    CONST robtarget Target_11220:=[[89.794609886,117.20347241,29.885035034],[0.692516726,0.060687774,-0.040025667,0.717729422],[0,0,0,0],[9E+09,9E+09,9E+09,9E+09,9E+09,9E+09]];
    CONST robtarget Target_11230:=[[90.590419724,116.924123639,29.863083326],[0.692516726,0.060687774,-0.040025666,0.717729422],[0,0,0,0],[9E+09,9E+09,9E+09,9E+09,9E+09,9E+09]];
    CONST robtarget Target_11240:=[[91.356578481,116.571453419,29.841743496],[0.692516726,0.060687774,-0.040025667,0.717729422],[0,0,0,0],[9E+09,9E+09,9E+09,9E+09,9E+09,9E+09]];
    CONST robtarget Target_11250:=[[92.086353126,116.148561032,29.821203079],[0.692516726,0.060687774,-0.040025667,0.717729422],[0,0,0,0],[9E+09,9E+09,9E+09,9E+09,9E+09,9E+09]];
    CONST robtarget Target_11260:=[[92.773330372,115.659162869,29.801642586],[0.692516726,0.060687774,-0.040025666,0.717729422],[0,0,0,0],[9E+09,9E+09,9E+09,9E+09,9E+09,9E+09]];
    CONST robtarget Target_11270:=[[93.411473041,115.107559779,29.783233914],[0.692516726,0.060687774,-0.040025667,0.717729422],[0,0,0,0],[9E+09,9E+09,9E+09,9E+09,9E+09,9E+09]];
    CONST robtarget Target_11280:=[[93.995173109,114.498599271,29.76613884],[0.692516726,0.060687774,-0.040025666,0.717729422],[0,0,0,0],[9E+09,9E+09,9E+09,9E+09,9E+09,9E+09]];
    CONST robtarget Target_11290:=[[94.519301002,113.837632911,29.750507595],[0.692516726,0.060687774,-0.040025667,0.717729422],[0,0,0,0],[9E+09,9E+09,9E+09,9E+09,9E+09,9E+09]];
    CONST robtarget Target_11300:=[[94.979250663,113.130469294,29.736477548],[0.692516726,0.060687774,-0.040025666,0.717729422],[0,0,0,0],[9E+09,9E+09,9E+09,9E+09,9E+09,9E+09]];
    CONST robtarget Target_11310:=[[95.370980037,112.383323003,29.724171995],[0.692516726,0.060687774,-0.040025666,0.717729422],[0,0,0,0],[9E+09,9E+09,9E+09,9E+09,9E+09,9E+09]];
    CONST robtarget Target_11320:=[[95.691046596,111.602759982,29.713699078],[0.692516726,0.060687774,-0.040025666,0.717729422],[0,0,0,0],[9E+09,9E+09,9E+09,9E+09,9E+09,9E+09]];
    CONST robtarget Target_11330:=[[95.93663758,110.79563985,29.705150834],[0.692516726,0.060687774,-0.040025666,0.717729422],[0,0,0,0],[9E+09,9E+09,9E+09,9E+09,9E+09,9E+09]];
    CONST robtarget Target_11340:=[[96.105594728,109.969055606,29.698602383],[0.692516726,0.060687774,-0.040025667,0.717729422],[0,0,0,0],[9E+09,9E+09,9E+09,9E+09,9E+09,9E+09]];
    CONST robtarget Target_11350:=[[96.196433238,109.130271302,29.694111275],[0.692516726,0.060687774,-0.040025667,0.717729422],[0,0,0,0],[9E+09,9E+09,9E+09,9E+09,9E+09,9E+09]];
    CONST robtarget Target_11360:=[[96.208354819,108.286658206,29.691716978],[0.692516726,0.060687774,-0.040025667,0.717729422],[0,0,0,0],[9E+09,9E+09,9E+09,9E+09,9E+09,9E+09]];
    CONST robtarget Target_11370:=[[96.141254703,107.445630019,29.691440532],[0.692516726,0.060687774,-0.040025667,0.717729422],[0,0,0,0],[9E+09,9E+09,9E+09,9E+09,9E+09,9E+09]];
    CONST robtarget Target_11380:=[[95.995722568,106.614577729,29.693284368],[0.692516726,0.060687774,-0.040025667,0.717729422],[0,0,0,0],[9E+09,9E+09,9E+09,9E+09,9E+09,9E+09]];
    CONST robtarget Target_11390:=[[95.773037356,105.80080465,29.697232281],[0.692516726,0.060687774,-0.040025667,0.717729422],[0,0,0,0],[9E+09,9E+09,9E+09,9E+09,9E+09,9E+09]];
    CONST robtarget Target_11400:=[[95.475156032,105.011462252,29.703249576],[0.692516726,0.060687774,-0.040025667,0.717729422],[0,0,0,0],[9E+09,9E+09,9E+09,9E+09,9E+09,9E+09]];
    CONST robtarget Target_11410:=[[95.104696388,104.253487303,29.711283375],[0.692516726,0.060687774,-0.040025666,0.717729422],[0,0,0,0],[9E+09,9E+09,9E+09,9E+09,9E+09,9E+09]];
    CONST robtarget Target_11420:=[[94.664914038,103.533540915,29.721263075],[0.692516726,0.060687774,-0.040025667,0.717729422],[0,0,0,0],[9E+09,9E+09,9E+09,9E+09,9E+09,9E+09]];
    CONST robtarget Target_11430:=[[94.159673804,102.857950002,29.733100975],[0.692516726,0.060687774,-0.040025667,0.717729422],[0,0,0,0],[9E+09,9E+09,9E+09,9E+09,9E+09,9E+09]];
    CONST robtarget Target_11440:=[[93.593415754,102.232651681,29.746693042],[0.692516726,0.060687774,-0.040025667,0.717729422],[0,0,0,0],[9E+09,9E+09,9E+09,9E+09,9E+09,9E+09]];
    CONST robtarget Target_11450:=[[92.971116187,101.663141097,29.761919829],[0.692516726,0.060687774,-0.040025666,0.717729422],[0,0,0,0],[9E+09,9E+09,9E+09,9E+09,9E+09,9E+09]];
    CONST robtarget Target_11460:=[[92.298243892,101.154423128,29.778647523],[0.692516726,0.060687774,-0.040025667,0.717729422],[0,0,0,0],[9E+09,9E+09,9E+09,9E+09,9E+09,9E+09]];
    CONST robtarget Target_11470:=[[91.580712095,100.710968408,29.79672912],[0.692516726,0.060687774,-0.040025667,0.717729422],[0,0,0,0],[9E+09,9E+09,9E+09,9E+09,9E+09,9E+09]];
    CONST robtarget Target_11480:=[[90.824826492,100.336674031,29.816005718],[0.692516726,0.060687774,-0.040025667,0.717729422],[0,0,0,0],[9E+09,9E+09,9E+09,9E+09,9E+09,9E+09]];
    CONST robtarget Target_11490:=[[90.037229833,100.034829312,29.836307913],[0.692516726,0.060687774,-0.040025667,0.717729422],[0,0,0,0],[9E+09,9E+09,9E+09,9E+09,9E+09,9E+09]];
    CONST robtarget Target_11500:=[[89.224843544,99.808086869,29.85745729],[0.692516726,0.060687774,-0.040025666,0.717729422],[0,0,0,0],[9E+09,9E+09,9E+09,9E+09,9E+09,9E+09]];
    CONST robtarget Target_11510:=[[88.394806907,99.658439327,29.879267987],[0.692516726,0.060687774,-0.040025666,0.717729422],[0,0,0,0],[9E+09,9E+09,9E+09,9E+09,9E+09,9E+09]];
    CONST robtarget Target_11520:=[[87.554414313,99.587201792,29.901548331],[0.692516726,0.060687774,-0.040025667,0.717729422],[0,0,0,0],[9E+09,9E+09,9E+09,9E+09,9E+09,9E+09]];
    CONST robtarget Target_11530:=[[86.753090736,99.66099158,-0.087656987],[0.692516726,0.060687774,-0.040025667,0.717729422],[0,0,0,0],[9E+09,9E+09,9E+09,9E+09,9E+09,9E+09]];
    CONST robtarget Target_11540:=[[119.551173325,78.726504599,-1.015545136],[0.692516726,0.060687774,-0.040025666,0.717729422],[0,0,0,0],[9E+09,9E+09,9E+09,9E+09,9E+09,9E+09]];
    CONST robtarget Target_11550:=[[120.352496902,78.652714811,28.973660182],[0.692516726,0.060687774,-0.040025666,0.717729422],[0,0,0,0],[9E+09,9E+09,9E+09,9E+09,9E+09,9E+09]];
    CONST robtarget Target_11560:=[[120.164706446,83.64915705,28.990971989],[0.692516726,0.060687774,-0.040025666,0.717729422],[0,0,0,0],[9E+09,9E+09,9E+09,9E+09,9E+09,9E+09]];
    CONST robtarget Target_11570:=[[110.175332474,83.272786458,29.256965985],[0.692516726,0.060687774,-0.040025666,0.717729422],[0,0,0,0],[9E+09,9E+09,9E+09,9E+09,9E+09,9E+09]];
    CONST robtarget Target_11580:=[[110.363122929,78.276344219,29.239654179],[0.692516726,0.060687774,-0.040025666,0.717729422],[0,0,0,0],[9E+09,9E+09,9E+09,9E+09,9E+09,9E+09]];
    CONST robtarget Target_11590:=[[120.352496902,78.652714811,28.973660182],[0.692516726,0.060687774,-0.040025666,0.717729422],[0,0,0,0],[9E+09,9E+09,9E+09,9E+09,9E+09,9E+09]];
    CONST robtarget Target_11600:=[[119.551173325,78.726504599,-1.015545136],[0.692516726,0.060687774,-0.040025666,0.717729422],[0,0,0,0],[9E+09,9E+09,9E+09,9E+09,9E+09,9E+09]];
    CONST robtarget Target_11610:=[[94.577738392,77.785578119,-0.350560144],[0.692516726,0.060687774,-0.040025666,0.717729422],[0,0,0,0],[9E+09,9E+09,9E+09,9E+09,9E+09,9E+09]];
    CONST robtarget Target_11620:=[[95.379061969,77.711788331,29.638645173],[0.692516726,0.060687774,-0.040025666,0.717729422],[0,0,0,0],[9E+09,9E+09,9E+09,9E+09,9E+09,9E+09]];
    CONST robtarget Target_11630:=[[105.368435942,78.088158923,29.372651177],[0.692516726,0.060687774,-0.040025666,0.717729422],[0,0,0,0],[9E+09,9E+09,9E+09,9E+09,9E+09,9E+09]];
    CONST robtarget Target_11640:=[[105.180645487,83.084601162,29.389962984],[0.692516726,0.060687774,-0.040025666,0.717729422],[0,0,0,0],[9E+09,9E+09,9E+09,9E+09,9E+09,9E+09]];
    CONST robtarget Target_11650:=[[95.191271514,82.70823057,29.65595698],[0.692516726,0.060687774,-0.040025666,0.717729422],[0,0,0,0],[9E+09,9E+09,9E+09,9E+09,9E+09,9E+09]];
    CONST robtarget Target_11660:=[[95.379061969,77.711788331,29.638645173],[0.692516726,0.060687774,-0.040025666,0.717729422],[0,0,0,0],[9E+09,9E+09,9E+09,9E+09,9E+09,9E+09]];
    CONST robtarget Target_11670:=[[94.577738392,77.785578119,-0.350560144],[0.692516726,0.060687774,-0.040025666,0.717729422],[0,0,0,0],[9E+09,9E+09,9E+09,9E+09,9E+09,9E+09]];
    CONST robtarget Target_11680:=[[89.583051406,77.597392823,-0.217563146],[0.692516726,0.060687774,-0.040025666,0.717729422],[0,0,0,0],[9E+09,9E+09,9E+09,9E+09,9E+09,9E+09]];
    CONST robtarget Target_11690:=[[90.384374983,77.523603036,29.771642172],[0.692516726,0.060687774,-0.040025666,0.717729422],[0,0,0,0],[9E+09,9E+09,9E+09,9E+09,9E+09,9E+09]];
    CONST robtarget Target_11700:=[[90.196584528,82.520045274,29.788953979],[0.692516726,0.060687774,-0.040025666,0.717729422],[0,0,0,0],[9E+09,9E+09,9E+09,9E+09,9E+09,9E+09]];
    CONST robtarget Target_11710:=[[80.207210555,82.143674683,30.054947975],[0.692516726,0.060687774,-0.040025666,0.717729422],[0,0,0,0],[9E+09,9E+09,9E+09,9E+09,9E+09,9E+09]];
    CONST robtarget Target_11720:=[[80.39500101,77.147232444,30.037636168],[0.692516726,0.060687774,-0.040025666,0.717729422],[0,0,0,0],[9E+09,9E+09,9E+09,9E+09,9E+09,9E+09]];
    CONST robtarget Target_11730:=[[90.384374983,77.523603036,29.771642172],[0.692516726,0.060687774,-0.040025666,0.717729422],[0,0,0,0],[9E+09,9E+09,9E+09,9E+09,9E+09,9E+09]];
    CONST robtarget Target_11740:=[[89.583051406,77.597392823,-0.217563146],[0.692516726,0.060687774,-0.040025666,0.717729422],[0,0,0,0],[9E+09,9E+09,9E+09,9E+09,9E+09,9E+09]];






    CONST jointtarget Home_ABS:= [[0,0,0,0,30,0],[9E+09,9E+09,9E+09,9E+09,9E+09,9E+09]];
    CONST jointtarget Mantenimiento_Point:= [[90,0,0,0,30,0],[9E+09,9E+09,9E+09,9E+09,9E+09,9E+09]];
    !***********************************************************
    !
    ! M?dulo:  Module1
    !
    ! Descripción:
    !   <Introduzca la descripción aquí>
    !
    ! Autor: pache
    !
    ! Versión: 1.0
    !
    !***********************************************************


    !***********************************************************
    !
    ! Procedimiento Main
    !
    !   Este es el punto de entrada de su programa
    !
PROC main()

        ! Limpiamos la pantalla del control virtual
        TPErase;
        TPWrite "SISTEMA INICIADO";

        MoveAbsJ Home_ABS, v300, z1, tool0;

        TPWrite "INICIO PROGRAMA";
        TPWrite "APAGADO BANDA TRANASPORTADORA";
        Reset DO_02;
        Reset DO_01;
        RESET BWD_Conveyor;
        RESET FWD_Conveyor;




        ! 1. Apagamos la banda por seguridad al arrancar

        WHILE TRUE DO

            IF DI_03 = 1 THEN
                Set BWD_Conveyor;
                WaitTime 4.275;
                Reset FWD_Conveyor;
                Reset BWD_Conveyor;
            ENDIF


            TPWrite "ESPERANDO QUE PRESIONE DI_01...";
            ! 2. Esperamos el botón de inicio
            IF DI_01 = 1 AND DI_02 = 0 THEN




                    TPWrite "MOVIENDO CAJA...";

                    ! 3. Encendemos la banda
                    set FWD_Conveyor;
                    set DO_01;

                    ! 4. Tiempo de viaje (ajustado a tu prueba)
                    WaitTime 4.275;

                    ! 5. Detenemos la caja
                    Reset FWD_Conveyor;
                    TPWrite "CAJA EN POSICION - INICIANDO GRABADO";

                    ! --------------------------------------------------------
                    ! 6. LLAMADA A LAS TRAYECTORIAS
                    Path_aprox;
                    WaitTime 1;
                    Path_duvan;
                    Path_mora;
                    Path_gusta;
                    Path_robot;
                    Path_220;
                    WaitTime 2;
                    Path_home;
                    WaitTime 5;
                    reset DO_01;

                ELSEIF DI_01 = 0 AND DI_02=1 THEN
                Set DO_02;
                TPWrite "RUTINA CAMBIO DE HERRAMIENTA";
                MoveAbsJ Mantenimiento_Point,v100,z1,tool0;
                TPWrite "PELIGRO";
                TPWrite "OPERARIO CERCA A HERRAMIENTA";
                TPWrite "PRESIONE LOS DOS BOTONES PARA CONTINUAR EL PROGRAMA";
                WaitDI DI_01,1;
                WaitDI DI_02,1;
                Reset DO_02;
                TPWrite "REANUDANDO PROGRAMA";
                WaitTime 3;
                MoveAbsJ Home_ABS,v100,z1,tool0;
                ELSEIF DI_01 = 0 AND DI_02=0 THEN
                TPWrite "ESPERANDO INSTRUCCIÓNES";
                ELSEIF DI_01 = 1 AND DI_02=1 THEN
                TPWrite "ERROR";
                TPWrite "NO DEBE PRESIONAR AMBAS ENTRADAS AL TIEMPO";
            ENDIF

            TPWrite "CICLO TERMINADO. MUEVA LA CAJA AL INICIO.";
        ENDWHILE
        WaitTime 1.0;
    ENDPROC




    PROC Path_aprox()
        MoveL Target_home,v100,z1,MarcadorVirtual\WObj:=wobj0;
        MoveL Target_aprox1,v100,z1,MarcadorVirtual\WObj:=wobj0;
        MoveL Target_aprox2,v100,z1,MarcadorVirtual\WObj:=wobj0;

    ENDPROC
    PROC Path_10()
        MoveL Target_aprox2,v60,z1,MarcadorVirtual\WObj:=wobj0;
        MoveL Target_10,v60,z1,MarcadorVirtual\WObj:=wobj_JMora;
    ENDPROC
    PROC Path_20()
        MoveL Target_540,v60,z1,MarcadorVirtual\WObj:=wobj_JMora;
        MoveL Target_550,v60,z1,MarcadorVirtual\WObj:=wobj_JMora;
    ENDPROC
    PROC Path_home()
        MoveL Target_home,v100,z1,MarcadorVirtual\WObj:=wobj0;
    ENDPROC
    PROC Path_30()
        MoveL Target_1070,v60,z1,MarcadorVirtual\WObj:=wobj_JMora;
        MoveL Target_1080,v60,z1,MarcadorVirtual\WObj:=wobj_JMora;
    ENDPROC
    PROC Path_40()
        MoveL Target_1560,v60,z1,MarcadorVirtual\WObj:=wobj_JMora;
        MoveL Target_1570,v60,z1,MarcadorVirtual\WObj:=wobj_JMora;
    ENDPROC
    PROC Path_50()
        MoveL Target_2360,v60,z1,MarcadorVirtual\WObj:=wobj_JMora;
        MoveL Target_2370,v60,z1,MarcadorVirtual\WObj:=wobj_JMora;
    ENDPROC
    PROC Path_60()
        MoveL Target_1070,v60,z1,MarcadorVirtual\WObj:=wobj_JMora;
        MoveL Target_1080,v60,z1,MarcadorVirtual\WObj:=wobj_JMora;
    ENDPROC
    PROC Path_D()
        MoveL Target_10,v60,z1,MarcadorVirtual\WObj:=wobj_JMora;
        MoveL Target_20,v60,z1,MarcadorVirtual\WObj:=wobj_JMora;
        MoveL Target_30,v60,z1,MarcadorVirtual\WObj:=wobj_JMora;
        MoveL Target_40,v60,z1,MarcadorVirtual\WObj:=wobj_JMora;
        MoveL Target_50,v60,z1,MarcadorVirtual\WObj:=wobj_JMora;
        MoveL Target_60,v60,z1,MarcadorVirtual\WObj:=wobj_JMora;
        MoveL Target_70,v60,z1,MarcadorVirtual\WObj:=wobj_JMora;
        MoveL Target_80,v60,z1,MarcadorVirtual\WObj:=wobj_JMora;
        MoveL Target_90,v60,z1,MarcadorVirtual\WObj:=wobj_JMora;
        MoveL Target_100,v60,z1,MarcadorVirtual\WObj:=wobj_JMora;
        MoveL Target_110,v60,z1,MarcadorVirtual\WObj:=wobj_JMora;
        MoveL Target_120,v60,z1,MarcadorVirtual\WObj:=wobj_JMora;
        MoveL Target_130,v60,z1,MarcadorVirtual\WObj:=wobj_JMora;
        MoveL Target_140,v60,z1,MarcadorVirtual\WObj:=wobj_JMora;
        MoveL Target_150,v60,z1,MarcadorVirtual\WObj:=wobj_JMora;
        MoveL Target_160,v60,z1,MarcadorVirtual\WObj:=wobj_JMora;
        MoveL Target_170,v60,z1,MarcadorVirtual\WObj:=wobj_JMora;
        MoveL Target_180,v60,z1,MarcadorVirtual\WObj:=wobj_JMora;
        MoveL Target_190,v60,z1,MarcadorVirtual\WObj:=wobj_JMora;
        MoveL Target_200,v60,z1,MarcadorVirtual\WObj:=wobj_JMora;
        MoveL Target_210,v60,z1,MarcadorVirtual\WObj:=wobj_JMora;
        MoveL Target_220,v60,z1,MarcadorVirtual\WObj:=wobj_JMora;
        MoveL Target_230,v60,z1,MarcadorVirtual\WObj:=wobj_JMora;
        MoveL Target_240,v60,z1,MarcadorVirtual\WObj:=wobj_JMora;
        MoveL Target_250,v60,z1,MarcadorVirtual\WObj:=wobj_JMora;
        MoveL Target_260,v60,z1,MarcadorVirtual\WObj:=wobj_JMora;
        MoveL Target_270,v60,z1,MarcadorVirtual\WObj:=wobj_JMora;
        MoveL Target_280,v60,z1,MarcadorVirtual\WObj:=wobj_JMora;
        MoveL Target_290,v60,z1,MarcadorVirtual\WObj:=wobj_JMora;
        MoveL Target_300,v60,z1,MarcadorVirtual\WObj:=wobj_JMora;
        MoveL Target_310,v60,z1,MarcadorVirtual\WObj:=wobj_JMora;
        MoveL Target_320,v60,z1,MarcadorVirtual\WObj:=wobj_JMora;
        MoveL Target_330,v60,z1,MarcadorVirtual\WObj:=wobj_JMora;
        MoveL Target_340,v60,z1,MarcadorVirtual\WObj:=wobj_JMora;
        MoveL Target_350,v60,z1,MarcadorVirtual\WObj:=wobj_JMora;
        MoveL Target_360,v60,z1,MarcadorVirtual\WObj:=wobj_JMora;
        MoveL Target_370,v60,z1,MarcadorVirtual\WObj:=wobj_JMora;
        MoveL Target_380,v60,z1,MarcadorVirtual\WObj:=wobj_JMora;
        MoveL Target_390,v60,z1,MarcadorVirtual\WObj:=wobj_JMora;
        MoveL Target_400,v60,z1,MarcadorVirtual\WObj:=wobj_JMora;
        MoveL Target_410,v60,z1,MarcadorVirtual\WObj:=wobj_JMora;
        MoveL Target_420,v60,z1,MarcadorVirtual\WObj:=wobj_JMora;
        MoveL Target_430,v60,z1,MarcadorVirtual\WObj:=wobj_JMora;
        MoveL Target_440,v60,z1,MarcadorVirtual\WObj:=wobj_JMora;
        MoveL Target_450,v60,z1,MarcadorVirtual\WObj:=wobj_JMora;
        MoveL Target_460,v60,z1,MarcadorVirtual\WObj:=wobj_JMora;
        MoveL Target_470,v60,z1,MarcadorVirtual\WObj:=wobj_JMora;
        MoveL Target_480,v60,z1,MarcadorVirtual\WObj:=wobj_JMora;
        MoveL Target_490,v60,z1,MarcadorVirtual\WObj:=wobj_JMora;
        MoveL Target_500,v60,z1,MarcadorVirtual\WObj:=wobj_JMora;
        MoveL Target_510,v60,z1,MarcadorVirtual\WObj:=wobj_JMora;
        MoveL Target_520,v60,z1,MarcadorVirtual\WObj:=wobj_JMora;
        MoveL Target_530,v60,z1,MarcadorVirtual\WObj:=wobj_JMora;
        MoveL Target_540,v60,z1,MarcadorVirtual\WObj:=wobj_JMora;
    ENDPROC
    PROC Path_U1()
        MoveL Target_550,v60,z1,MarcadorVirtual\WObj:=wobj_JMora;
        MoveL Target_560,v60,z1,MarcadorVirtual\WObj:=wobj_JMora;
        MoveL Target_570,v60,z1,MarcadorVirtual\WObj:=wobj_JMora;
        MoveL Target_580,v60,z1,MarcadorVirtual\WObj:=wobj_JMora;
        MoveL Target_590,v60,z1,MarcadorVirtual\WObj:=wobj_JMora;
        MoveL Target_600,v60,z1,MarcadorVirtual\WObj:=wobj_JMora;
        MoveL Target_610,v60,z1,MarcadorVirtual\WObj:=wobj_JMora;
        MoveL Target_620,v60,z1,MarcadorVirtual\WObj:=wobj_JMora;
        MoveL Target_630,v60,z1,MarcadorVirtual\WObj:=wobj_JMora;
        MoveL Target_640,v60,z1,MarcadorVirtual\WObj:=wobj_JMora;
        MoveL Target_650,v60,z1,MarcadorVirtual\WObj:=wobj_JMora;
        MoveL Target_660,v60,z1,MarcadorVirtual\WObj:=wobj_JMora;
        MoveL Target_670,v60,z1,MarcadorVirtual\WObj:=wobj_JMora;
        MoveL Target_680,v60,z1,MarcadorVirtual\WObj:=wobj_JMora;
        MoveL Target_690,v60,z1,MarcadorVirtual\WObj:=wobj_JMora;
        MoveL Target_700,v60,z1,MarcadorVirtual\WObj:=wobj_JMora;
        MoveL Target_710,v60,z1,MarcadorVirtual\WObj:=wobj_JMora;
        MoveL Target_720,v60,z1,MarcadorVirtual\WObj:=wobj_JMora;
        MoveL Target_730,v60,z1,MarcadorVirtual\WObj:=wobj_JMora;
        MoveL Target_740,v60,z1,MarcadorVirtual\WObj:=wobj_JMora;
        MoveL Target_750,v60,z1,MarcadorVirtual\WObj:=wobj_JMora;
        MoveL Target_760,v60,z1,MarcadorVirtual\WObj:=wobj_JMora;
        MoveL Target_770,v60,z1,MarcadorVirtual\WObj:=wobj_JMora;
        MoveL Target_780,v60,z1,MarcadorVirtual\WObj:=wobj_JMora;
        MoveL Target_790,v60,z1,MarcadorVirtual\WObj:=wobj_JMora;
        MoveL Target_800,v60,z1,MarcadorVirtual\WObj:=wobj_JMora;
        MoveL Target_810,v60,z1,MarcadorVirtual\WObj:=wobj_JMora;
        MoveL Target_820,v60,z1,MarcadorVirtual\WObj:=wobj_JMora;
        MoveL Target_830,v60,z1,MarcadorVirtual\WObj:=wobj_JMora;
        MoveL Target_840,v60,z1,MarcadorVirtual\WObj:=wobj_JMora;
        MoveL Target_850,v60,z1,MarcadorVirtual\WObj:=wobj_JMora;
        MoveL Target_860,v60,z1,MarcadorVirtual\WObj:=wobj_JMora;
        MoveL Target_870,v60,z1,MarcadorVirtual\WObj:=wobj_JMora;
        MoveL Target_880,v60,z1,MarcadorVirtual\WObj:=wobj_JMora;
        MoveL Target_890,v60,z1,MarcadorVirtual\WObj:=wobj_JMora;
        MoveL Target_900,v60,z1,MarcadorVirtual\WObj:=wobj_JMora;
        MoveL Target_910,v60,z1,MarcadorVirtual\WObj:=wobj_JMora;
        MoveL Target_920,v60,z1,MarcadorVirtual\WObj:=wobj_JMora;
        MoveL Target_930,v60,z1,MarcadorVirtual\WObj:=wobj_JMora;
        MoveL Target_940,v60,z1,MarcadorVirtual\WObj:=wobj_JMora;
        MoveL Target_950,v60,z1,MarcadorVirtual\WObj:=wobj_JMora;
        MoveL Target_960,v60,z1,MarcadorVirtual\WObj:=wobj_JMora;
        MoveL Target_970,v60,z1,MarcadorVirtual\WObj:=wobj_JMora;
        MoveL Target_980,v60,z1,MarcadorVirtual\WObj:=wobj_JMora;
        MoveL Target_990,v60,z1,MarcadorVirtual\WObj:=wobj_JMora;
        MoveL Target_1000,v60,z1,MarcadorVirtual\WObj:=wobj_JMora;
        MoveL Target_1010,v60,z1,MarcadorVirtual\WObj:=wobj_JMora;
        MoveL Target_1020,v60,z1,MarcadorVirtual\WObj:=wobj_JMora;
        MoveL Target_1030,v60,z1,MarcadorVirtual\WObj:=wobj_JMora;
        MoveL Target_1040,v60,z1,MarcadorVirtual\WObj:=wobj_JMora;
        MoveL Target_1050,v60,z1,MarcadorVirtual\WObj:=wobj_JMora;
        MoveL Target_1060,v60,z1,MarcadorVirtual\WObj:=wobj_JMora;
        MoveL Target_1070,v60,z1,MarcadorVirtual\WObj:=wobj_JMora;
    ENDPROC
    PROC Path_V()
        MoveL Target_1080,v60,z1,MarcadorVirtual\WObj:=wobj_JMora;
        MoveL Target_1090,v60,z1,MarcadorVirtual\WObj:=wobj_JMora;
        MoveL Target_1100,v60,z1,MarcadorVirtual\WObj:=wobj_JMora;
        MoveL Target_1110,v60,z1,MarcadorVirtual\WObj:=wobj_JMora;
        MoveL Target_1120,v60,z1,MarcadorVirtual\WObj:=wobj_JMora;
        MoveL Target_1130,v60,z1,MarcadorVirtual\WObj:=wobj_JMora;
        MoveL Target_1140,v60,z1,MarcadorVirtual\WObj:=wobj_JMora;
        MoveL Target_1150,v60,z1,MarcadorVirtual\WObj:=wobj_JMora;
        MoveL Target_1160,v60,z1,MarcadorVirtual\WObj:=wobj_JMora;
        MoveL Target_1170,v60,z1,MarcadorVirtual\WObj:=wobj_JMora;
        MoveL Target_1180,v60,z1,MarcadorVirtual\WObj:=wobj_JMora;
        MoveL Target_1190,v60,z1,MarcadorVirtual\WObj:=wobj_JMora;
        MoveL Target_1200,v60,z1,MarcadorVirtual\WObj:=wobj_JMora;
        MoveL Target_1210,v60,z1,MarcadorVirtual\WObj:=wobj_JMora;
        MoveL Target_1220,v60,z1,MarcadorVirtual\WObj:=wobj_JMora;
        MoveL Target_1230,v60,z1,MarcadorVirtual\WObj:=wobj_JMora;
        MoveL Target_1240,v60,z1,MarcadorVirtual\WObj:=wobj_JMora;
        MoveL Target_1250,v60,z1,MarcadorVirtual\WObj:=wobj_JMora;
        MoveL Target_1260,v60,z1,MarcadorVirtual\WObj:=wobj_JMora;
        MoveL Target_1270,v60,z1,MarcadorVirtual\WObj:=wobj_JMora;
        MoveL Target_1280,v60,z1,MarcadorVirtual\WObj:=wobj_JMora;
        MoveL Target_1290,v60,z1,MarcadorVirtual\WObj:=wobj_JMora;
        MoveL Target_1300,v60,z1,MarcadorVirtual\WObj:=wobj_JMora;
        MoveL Target_1310,v60,z1,MarcadorVirtual\WObj:=wobj_JMora;
        MoveL Target_1320,v60,z1,MarcadorVirtual\WObj:=wobj_JMora;
        MoveL Target_1330,v60,z1,MarcadorVirtual\WObj:=wobj_JMora;
        MoveL Target_1340,v60,z1,MarcadorVirtual\WObj:=wobj_JMora;
        MoveL Target_1350,v60,z1,MarcadorVirtual\WObj:=wobj_JMora;
        MoveL Target_1360,v60,z1,MarcadorVirtual\WObj:=wobj_JMora;
        MoveL Target_1370,v60,z1,MarcadorVirtual\WObj:=wobj_JMora;
        MoveL Target_1380,v60,z1,MarcadorVirtual\WObj:=wobj_JMora;
        MoveL Target_1390,v60,z1,MarcadorVirtual\WObj:=wobj_JMora;
        MoveL Target_1400,v60,z1,MarcadorVirtual\WObj:=wobj_JMora;
        MoveL Target_1410,v60,z1,MarcadorVirtual\WObj:=wobj_JMora;
        MoveL Target_1420,v60,z1,MarcadorVirtual\WObj:=wobj_JMora;
        MoveL Target_1430,v60,z1,MarcadorVirtual\WObj:=wobj_JMora;
        MoveL Target_1440,v60,z1,MarcadorVirtual\WObj:=wobj_JMora;
        MoveL Target_1450,v60,z1,MarcadorVirtual\WObj:=wobj_JMora;
        MoveL Target_1460,v60,z1,MarcadorVirtual\WObj:=wobj_JMora;
        MoveL Target_1470,v60,z1,MarcadorVirtual\WObj:=wobj_JMora;
        MoveL Target_1480,v60,z1,MarcadorVirtual\WObj:=wobj_JMora;
        MoveL Target_1490,v60,z1,MarcadorVirtual\WObj:=wobj_JMora;
        MoveL Target_1500,v60,z1,MarcadorVirtual\WObj:=wobj_JMora;
        MoveL Target_1510,v60,z1,MarcadorVirtual\WObj:=wobj_JMora;
        MoveL Target_1520,v60,z1,MarcadorVirtual\WObj:=wobj_JMora;
        MoveL Target_1530,v60,z1,MarcadorVirtual\WObj:=wobj_JMora;
        MoveL Target_1540,v60,z1,MarcadorVirtual\WObj:=wobj_JMora;
        MoveL Target_1550,v60,z1,MarcadorVirtual\WObj:=wobj_JMora;
        MoveL Target_1560,v60,z1,MarcadorVirtual\WObj:=wobj_JMora;
    ENDPROC
    PROC Path_A1()
        MoveL Target_1570,v60,z1,MarcadorVirtual\WObj:=wobj_JMora;
        MoveL Target_1580,v60,z1,MarcadorVirtual\WObj:=wobj_JMora;
        MoveL Target_1590,v60,z1,MarcadorVirtual\WObj:=wobj_JMora;
        MoveL Target_1600,v60,z1,MarcadorVirtual\WObj:=wobj_JMora;
        MoveL Target_1610,v60,z1,MarcadorVirtual\WObj:=wobj_JMora;
        MoveL Target_1620,v60,z1,MarcadorVirtual\WObj:=wobj_JMora;
        MoveL Target_1630,v60,z1,MarcadorVirtual\WObj:=wobj_JMora;
        MoveL Target_1640,v60,z1,MarcadorVirtual\WObj:=wobj_JMora;
        MoveL Target_1650,v60,z1,MarcadorVirtual\WObj:=wobj_JMora;
        MoveL Target_1660,v60,z1,MarcadorVirtual\WObj:=wobj_JMora;
        MoveL Target_1670,v60,z1,MarcadorVirtual\WObj:=wobj_JMora;
        MoveL Target_1680,v60,z1,MarcadorVirtual\WObj:=wobj_JMora;
        MoveL Target_1690,v60,z1,MarcadorVirtual\WObj:=wobj_JMora;
        MoveL Target_1700,v60,z1,MarcadorVirtual\WObj:=wobj_JMora;
        MoveL Target_1710,v60,z1,MarcadorVirtual\WObj:=wobj_JMora;
        MoveL Target_1720,v60,z1,MarcadorVirtual\WObj:=wobj_JMora;
        MoveL Target_1730,v60,z1,MarcadorVirtual\WObj:=wobj_JMora;
        MoveL Target_1740,v60,z1,MarcadorVirtual\WObj:=wobj_JMora;
        MoveL Target_1750,v60,z1,MarcadorVirtual\WObj:=wobj_JMora;
        MoveL Target_1760,v60,z1,MarcadorVirtual\WObj:=wobj_JMora;
        MoveL Target_1770,v60,z1,MarcadorVirtual\WObj:=wobj_JMora;
        MoveL Target_1780,v60,z1,MarcadorVirtual\WObj:=wobj_JMora;
        MoveL Target_1790,v60,z1,MarcadorVirtual\WObj:=wobj_JMora;
        MoveL Target_1800,v60,z1,MarcadorVirtual\WObj:=wobj_JMora;
        MoveL Target_1810,v60,z1,MarcadorVirtual\WObj:=wobj_JMora;
        MoveL Target_1820,v60,z1,MarcadorVirtual\WObj:=wobj_JMora;
        MoveL Target_1830,v60,z1,MarcadorVirtual\WObj:=wobj_JMora;
        MoveL Target_1840,v60,z1,MarcadorVirtual\WObj:=wobj_JMora;
        MoveL Target_1850,v60,z1,MarcadorVirtual\WObj:=wobj_JMora;
        MoveL Target_1860,v60,z1,MarcadorVirtual\WObj:=wobj_JMora;
        MoveL Target_1870,v60,z1,MarcadorVirtual\WObj:=wobj_JMora;
        MoveL Target_1880,v60,z1,MarcadorVirtual\WObj:=wobj_JMora;
        MoveL Target_1890,v60,z1,MarcadorVirtual\WObj:=wobj_JMora;
        MoveL Target_1900,v60,z1,MarcadorVirtual\WObj:=wobj_JMora;
        MoveL Target_1910,v60,z1,MarcadorVirtual\WObj:=wobj_JMora;
        MoveL Target_1920,v60,z1,MarcadorVirtual\WObj:=wobj_JMora;
        MoveL Target_1930,v60,z1,MarcadorVirtual\WObj:=wobj_JMora;
        MoveL Target_1940,v60,z1,MarcadorVirtual\WObj:=wobj_JMora;
        MoveL Target_1950,v60,z1,MarcadorVirtual\WObj:=wobj_JMora;
        MoveL Target_1960,v60,z1,MarcadorVirtual\WObj:=wobj_JMora;
        MoveL Target_1970,v60,z1,MarcadorVirtual\WObj:=wobj_JMora;
        MoveL Target_1980,v60,z1,MarcadorVirtual\WObj:=wobj_JMora;
        MoveL Target_1990,v60,z1,MarcadorVirtual\WObj:=wobj_JMora;
        MoveL Target_2000,v60,z1,MarcadorVirtual\WObj:=wobj_JMora;
        MoveL Target_2010,v60,z1,MarcadorVirtual\WObj:=wobj_JMora;
        MoveL Target_2020,v60,z1,MarcadorVirtual\WObj:=wobj_JMora;
        MoveL Target_2030,v60,z1,MarcadorVirtual\WObj:=wobj_JMora;
        MoveL Target_2040,v60,z1,MarcadorVirtual\WObj:=wobj_JMora;
        MoveL Target_2050,v60,z1,MarcadorVirtual\WObj:=wobj_JMora;
        MoveL Target_2060,v60,z1,MarcadorVirtual\WObj:=wobj_JMora;
        MoveL Target_2070,v60,z1,MarcadorVirtual\WObj:=wobj_JMora;
        MoveL Target_2080,v60,z1,MarcadorVirtual\WObj:=wobj_JMora;
        MoveL Target_2090,v60,z1,MarcadorVirtual\WObj:=wobj_JMora;
        MoveL Target_2100,v60,z1,MarcadorVirtual\WObj:=wobj_JMora;
        MoveL Target_2110,v60,z1,MarcadorVirtual\WObj:=wobj_JMora;
        MoveL Target_2120,v60,z1,MarcadorVirtual\WObj:=wobj_JMora;
        MoveL Target_2130,v60,z1,MarcadorVirtual\WObj:=wobj_JMora;
        MoveL Target_2140,v60,z1,MarcadorVirtual\WObj:=wobj_JMora;
        MoveL Target_2150,v60,z1,MarcadorVirtual\WObj:=wobj_JMora;
        MoveL Target_2160,v60,z1,MarcadorVirtual\WObj:=wobj_JMora;
        MoveL Target_2170,v60,z1,MarcadorVirtual\WObj:=wobj_JMora;
        MoveL Target_2180,v60,z1,MarcadorVirtual\WObj:=wobj_JMora;
        MoveL Target_2190,v60,z1,MarcadorVirtual\WObj:=wobj_JMora;
        MoveL Target_2200,v60,z1,MarcadorVirtual\WObj:=wobj_JMora;
        MoveL Target_2210,v60,z1,MarcadorVirtual\WObj:=wobj_JMora;
        MoveL Target_2220,v60,z1,MarcadorVirtual\WObj:=wobj_JMora;
        MoveL Target_2230,v60,z1,MarcadorVirtual\WObj:=wobj_JMora;
        MoveL Target_2240,v60,z1,MarcadorVirtual\WObj:=wobj_JMora;
        MoveL Target_2250,v60,z1,MarcadorVirtual\WObj:=wobj_JMora;
        MoveL Target_2260,v60,z1,MarcadorVirtual\WObj:=wobj_JMora;
        MoveL Target_2270,v60,z1,MarcadorVirtual\WObj:=wobj_JMora;
        MoveL Target_2280,v60,z1,MarcadorVirtual\WObj:=wobj_JMora;
        MoveL Target_2290,v60,z1,MarcadorVirtual\WObj:=wobj_JMora;
        MoveL Target_2300,v60,z1,MarcadorVirtual\WObj:=wobj_JMora;
        MoveL Target_2310,v60,z1,MarcadorVirtual\WObj:=wobj_JMora;
        MoveL Target_2320,v60,z1,MarcadorVirtual\WObj:=wobj_JMora;
        MoveL Target_2330,v60,z1,MarcadorVirtual\WObj:=wobj_JMora;
        MoveL Target_2340,v60,z1,MarcadorVirtual\WObj:=wobj_JMora;
        MoveL Target_2350,v60,z1,MarcadorVirtual\WObj:=wobj_JMora;
        MoveL Target_2360,v60,z1,MarcadorVirtual\WObj:=wobj_JMora;
    ENDPROC
    PROC Path_N()
        MoveL Target_2370,v60,z1,MarcadorVirtual\WObj:=wobj_JMora;
        MoveL Target_2380,v60,z1,MarcadorVirtual\WObj:=wobj_JMora;
        MoveL Target_2390,v60,z1,MarcadorVirtual\WObj:=wobj_JMora;
        MoveL Target_2400,v60,z1,MarcadorVirtual\WObj:=wobj_JMora;
        MoveL Target_2410,v60,z1,MarcadorVirtual\WObj:=wobj_JMora;
        MoveL Target_2420,v60,z1,MarcadorVirtual\WObj:=wobj_JMora;
        MoveL Target_2430,v60,z1,MarcadorVirtual\WObj:=wobj_JMora;
        MoveL Target_2440,v60,z1,MarcadorVirtual\WObj:=wobj_JMora;
        MoveL Target_2450,v60,z1,MarcadorVirtual\WObj:=wobj_JMora;
        MoveL Target_2460,v60,z1,MarcadorVirtual\WObj:=wobj_JMora;
        MoveL Target_2470,v60,z1,MarcadorVirtual\WObj:=wobj_JMora;
        MoveL Target_2480,v60,z1,MarcadorVirtual\WObj:=wobj_JMora;
        MoveL Target_2490,v60,z1,MarcadorVirtual\WObj:=wobj_JMora;
        MoveL Target_2500,v60,z1,MarcadorVirtual\WObj:=wobj_JMora;
        MoveL Target_2510,v60,z1,MarcadorVirtual\WObj:=wobj_JMora;
        MoveL Target_2520,v60,z1,MarcadorVirtual\WObj:=wobj_JMora;
        MoveL Target_2530,v60,z1,MarcadorVirtual\WObj:=wobj_JMora;
        MoveL Target_2540,v60,z1,MarcadorVirtual\WObj:=wobj_JMora;
        MoveL Target_2550,v60,z1,MarcadorVirtual\WObj:=wobj_JMora;
        MoveL Target_2560,v60,z1,MarcadorVirtual\WObj:=wobj_JMora;
        MoveL Target_2570,v60,z1,MarcadorVirtual\WObj:=wobj_JMora;
        MoveL Target_2580,v60,z1,MarcadorVirtual\WObj:=wobj_JMora;
        MoveL Target_2590,v60,z1,MarcadorVirtual\WObj:=wobj_JMora;
        MoveL Target_2600,v60,z1,MarcadorVirtual\WObj:=wobj_JMora;
        MoveL Target_2610,v60,z1,MarcadorVirtual\WObj:=wobj_JMora;
        MoveL Target_2620,v60,z1,MarcadorVirtual\WObj:=wobj_JMora;
        MoveL Target_2630,v60,z1,MarcadorVirtual\WObj:=wobj_JMora;
        MoveL Target_2640,v60,z1,MarcadorVirtual\WObj:=wobj_JMora;
        MoveL Target_2650,v60,z1,MarcadorVirtual\WObj:=wobj_JMora;
        MoveL Target_2660,v60,z1,MarcadorVirtual\WObj:=wobj_JMora;
    ENDPROC


    PROC Path_duvan()
            Path_10;
            Path_D;
            Path_20;
            Path_U1;
            Path_30;
            Path_V;
            Path_40;
            Path_A1;
            Path_50;
            Path_N;
    ENDPROC

      PROC Path_mora()
            Path_70;
            Path_M;
            Path_80;
            Path_O;
            Path_90;
            Path_R;
            Path_100;
            Path_A2;
    ENDPROC



      PROC Path_gusta()
            Path_110;
            Path_G;
            Path_120;
            Path_U2;
            Path_130;
            Path_s;
            Path_140;
            Path_T;
            Path_150;
            Path_A3;
    ENDPROC


      PROC Path_robot()
            Path_160;
            Path_cara;
            Path_170;
            Path_ojo1;
            Path_180;
            Path_ojo2;
            Path_190;
            Path_boca1;
            Path_200;
            Path_boca2;
            Path_210;
            Path_boca3;
    ENDPROC
    PROC Path_M()
        MoveL Target_2670,v60,z1,MarcadorVirtual\WObj:=wobj_JMora;
        MoveL Target_2680,v60,z1,MarcadorVirtual\WObj:=wobj_JMora;
        MoveL Target_2690,v60,z1,MarcadorVirtual\WObj:=wobj_JMora;
        MoveL Target_2700,v60,z1,MarcadorVirtual\WObj:=wobj_JMora;
        MoveL Target_2710,v60,z1,MarcadorVirtual\WObj:=wobj_JMora;
        MoveL Target_2720,v60,z1,MarcadorVirtual\WObj:=wobj_JMora;
        MoveL Target_2730,v60,z1,MarcadorVirtual\WObj:=wobj_JMora;
        MoveL Target_2740,v60,z1,MarcadorVirtual\WObj:=wobj_JMora;
        MoveL Target_2750,v60,z1,MarcadorVirtual\WObj:=wobj_JMora;
        MoveL Target_2760,v60,z1,MarcadorVirtual\WObj:=wobj_JMora;
        MoveL Target_2770,v60,z1,MarcadorVirtual\WObj:=wobj_JMora;
        MoveL Target_2780,v60,z1,MarcadorVirtual\WObj:=wobj_JMora;
        MoveL Target_2790,v60,z1,MarcadorVirtual\WObj:=wobj_JMora;
        MoveL Target_2800,v60,z1,MarcadorVirtual\WObj:=wobj_JMora;
        MoveL Target_2810,v60,z1,MarcadorVirtual\WObj:=wobj_JMora;
        MoveL Target_2820,v60,z1,MarcadorVirtual\WObj:=wobj_JMora;
        MoveL Target_2830,v60,z1,MarcadorVirtual\WObj:=wobj_JMora;
        MoveL Target_2840,v60,z1,MarcadorVirtual\WObj:=wobj_JMora;
        MoveL Target_2850,v60,z1,MarcadorVirtual\WObj:=wobj_JMora;
        MoveL Target_2860,v60,z1,MarcadorVirtual\WObj:=wobj_JMora;
        MoveL Target_2870,v60,z1,MarcadorVirtual\WObj:=wobj_JMora;
        MoveL Target_2880,v60,z1,MarcadorVirtual\WObj:=wobj_JMora;
        MoveL Target_2890,v60,z1,MarcadorVirtual\WObj:=wobj_JMora;
        MoveL Target_2900,v60,z1,MarcadorVirtual\WObj:=wobj_JMora;
        MoveL Target_2910,v60,z1,MarcadorVirtual\WObj:=wobj_JMora;
        MoveL Target_2920,v60,z1,MarcadorVirtual\WObj:=wobj_JMora;
        MoveL Target_2930,v60,z1,MarcadorVirtual\WObj:=wobj_JMora;
        MoveL Target_2940,v60,z1,MarcadorVirtual\WObj:=wobj_JMora;
        MoveL Target_2950,v60,z1,MarcadorVirtual\WObj:=wobj_JMora;
        MoveL Target_2960,v60,z1,MarcadorVirtual\WObj:=wobj_JMora;
        MoveL Target_2970,v60,z1,MarcadorVirtual\WObj:=wobj_JMora;
        MoveL Target_2980,v60,z1,MarcadorVirtual\WObj:=wobj_JMora;
        MoveL Target_2990,v60,z1,MarcadorVirtual\WObj:=wobj_JMora;
        MoveL Target_3000,v60,z1,MarcadorVirtual\WObj:=wobj_JMora;
        MoveL Target_3010,v60,z1,MarcadorVirtual\WObj:=wobj_JMora;
        MoveL Target_3020,v60,z1,MarcadorVirtual\WObj:=wobj_JMora;
        MoveL Target_3030,v60,z1,MarcadorVirtual\WObj:=wobj_JMora;
        MoveL Target_3040,v60,z1,MarcadorVirtual\WObj:=wobj_JMora;
        MoveL Target_3050,v60,z1,MarcadorVirtual\WObj:=wobj_JMora;
        MoveL Target_3060,v60,z1,MarcadorVirtual\WObj:=wobj_JMora;
        MoveL Target_3070,v60,z1,MarcadorVirtual\WObj:=wobj_JMora;
        MoveL Target_3080,v60,z1,MarcadorVirtual\WObj:=wobj_JMora;
        MoveL Target_3090,v60,z1,MarcadorVirtual\WObj:=wobj_JMora;
        MoveL Target_3100,v60,z1,MarcadorVirtual\WObj:=wobj_JMora;
        MoveL Target_3110,v60,z1,MarcadorVirtual\WObj:=wobj_JMora;
        MoveL Target_3120,v60,z1,MarcadorVirtual\WObj:=wobj_JMora;
        MoveL Target_3130,v60,z1,MarcadorVirtual\WObj:=wobj_JMora;
    ENDPROC
    PROC Path_O()
        MoveL Target_3140,v60,z1,MarcadorVirtual\WObj:=wobj_JMora;
        MoveL Target_3150,v60,z1,MarcadorVirtual\WObj:=wobj_JMora;
        MoveL Target_3160,v60,z1,MarcadorVirtual\WObj:=wobj_JMora;
        MoveL Target_3170,v60,z1,MarcadorVirtual\WObj:=wobj_JMora;
        MoveL Target_3180,v60,z1,MarcadorVirtual\WObj:=wobj_JMora;
        MoveL Target_3190,v60,z1,MarcadorVirtual\WObj:=wobj_JMora;
        MoveL Target_3200,v60,z1,MarcadorVirtual\WObj:=wobj_JMora;
        MoveL Target_3210,v60,z1,MarcadorVirtual\WObj:=wobj_JMora;
        MoveL Target_3220,v60,z1,MarcadorVirtual\WObj:=wobj_JMora;
        MoveL Target_3230,v60,z1,MarcadorVirtual\WObj:=wobj_JMora;
        MoveL Target_3240,v60,z1,MarcadorVirtual\WObj:=wobj_JMora;
        MoveL Target_3250,v60,z1,MarcadorVirtual\WObj:=wobj_JMora;
        MoveL Target_3260,v60,z1,MarcadorVirtual\WObj:=wobj_JMora;
        MoveL Target_3270,v60,z1,MarcadorVirtual\WObj:=wobj_JMora;
        MoveL Target_3280,v60,z1,MarcadorVirtual\WObj:=wobj_JMora;
        MoveL Target_3290,v60,z1,MarcadorVirtual\WObj:=wobj_JMora;
        MoveL Target_3300,v60,z1,MarcadorVirtual\WObj:=wobj_JMora;
        MoveL Target_3310,v60,z1,MarcadorVirtual\WObj:=wobj_JMora;
        MoveL Target_3320,v60,z1,MarcadorVirtual\WObj:=wobj_JMora;
        MoveL Target_3330,v60,z1,MarcadorVirtual\WObj:=wobj_JMora;
        MoveL Target_3340,v60,z1,MarcadorVirtual\WObj:=wobj_JMora;
        MoveL Target_3350,v60,z1,MarcadorVirtual\WObj:=wobj_JMora;
        MoveL Target_3360,v60,z1,MarcadorVirtual\WObj:=wobj_JMora;
        MoveL Target_3370,v60,z1,MarcadorVirtual\WObj:=wobj_JMora;
        MoveL Target_3380,v60,z1,MarcadorVirtual\WObj:=wobj_JMora;
        MoveL Target_3390,v60,z1,MarcadorVirtual\WObj:=wobj_JMora;
        MoveL Target_3400,v60,z1,MarcadorVirtual\WObj:=wobj_JMora;
        MoveL Target_3410,v60,z1,MarcadorVirtual\WObj:=wobj_JMora;
        MoveL Target_3420,v60,z1,MarcadorVirtual\WObj:=wobj_JMora;
        MoveL Target_3430,v60,z1,MarcadorVirtual\WObj:=wobj_JMora;
        MoveL Target_3440,v60,z1,MarcadorVirtual\WObj:=wobj_JMora;
        MoveL Target_3450,v60,z1,MarcadorVirtual\WObj:=wobj_JMora;
        MoveL Target_3460,v60,z1,MarcadorVirtual\WObj:=wobj_JMora;
        MoveL Target_3470,v60,z1,MarcadorVirtual\WObj:=wobj_JMora;
        MoveL Target_3480,v60,z1,MarcadorVirtual\WObj:=wobj_JMora;
        MoveL Target_3490,v60,z1,MarcadorVirtual\WObj:=wobj_JMora;
        MoveL Target_3500,v60,z1,MarcadorVirtual\WObj:=wobj_JMora;
        MoveL Target_3510,v60,z1,MarcadorVirtual\WObj:=wobj_JMora;
        MoveL Target_3520,v60,z1,MarcadorVirtual\WObj:=wobj_JMora;
        MoveL Target_3530,v60,z1,MarcadorVirtual\WObj:=wobj_JMora;
        MoveL Target_3540,v60,z1,MarcadorVirtual\WObj:=wobj_JMora;
        MoveL Target_3550,v60,z1,MarcadorVirtual\WObj:=wobj_JMora;
        MoveL Target_3560,v60,z1,MarcadorVirtual\WObj:=wobj_JMora;
        MoveL Target_3570,v60,z1,MarcadorVirtual\WObj:=wobj_JMora;
        MoveL Target_3580,v60,z1,MarcadorVirtual\WObj:=wobj_JMora;
        MoveL Target_3590,v60,z1,MarcadorVirtual\WObj:=wobj_JMora;
        MoveL Target_3600,v60,z1,MarcadorVirtual\WObj:=wobj_JMora;
        MoveL Target_3610,v60,z1,MarcadorVirtual\WObj:=wobj_JMora;
        MoveL Target_3620,v60,z1,MarcadorVirtual\WObj:=wobj_JMora;
        MoveL Target_3630,v60,z1,MarcadorVirtual\WObj:=wobj_JMora;
        MoveL Target_3640,v60,z1,MarcadorVirtual\WObj:=wobj_JMora;
        MoveL Target_3650,v60,z1,MarcadorVirtual\WObj:=wobj_JMora;
        MoveL Target_3660,v60,z1,MarcadorVirtual\WObj:=wobj_JMora;
        MoveL Target_3670,v60,z1,MarcadorVirtual\WObj:=wobj_JMora;
        MoveL Target_3680,v60,z1,MarcadorVirtual\WObj:=wobj_JMora;
        MoveL Target_3690,v60,z1,MarcadorVirtual\WObj:=wobj_JMora;
        MoveL Target_3700,v60,z1,MarcadorVirtual\WObj:=wobj_JMora;
        MoveL Target_3710,v60,z1,MarcadorVirtual\WObj:=wobj_JMora;
        MoveL Target_3720,v60,z1,MarcadorVirtual\WObj:=wobj_JMora;
        MoveL Target_3730,v60,z1,MarcadorVirtual\WObj:=wobj_JMora;
        MoveL Target_3740,v60,z1,MarcadorVirtual\WObj:=wobj_JMora;
        MoveL Target_3750,v60,z1,MarcadorVirtual\WObj:=wobj_JMora;
        MoveL Target_3760,v60,z1,MarcadorVirtual\WObj:=wobj_JMora;
        MoveL Target_3770,v60,z1,MarcadorVirtual\WObj:=wobj_JMora;
        MoveL Target_3780,v60,z1,MarcadorVirtual\WObj:=wobj_JMora;
        MoveL Target_3790,v60,z1,MarcadorVirtual\WObj:=wobj_JMora;
        MoveL Target_3800,v60,z1,MarcadorVirtual\WObj:=wobj_JMora;
        MoveL Target_3810,v60,z1,MarcadorVirtual\WObj:=wobj_JMora;
        MoveL Target_3820,v60,z1,MarcadorVirtual\WObj:=wobj_JMora;
    ENDPROC
    PROC Path_R()
        MoveL Target_3830,v60,z1,MarcadorVirtual\WObj:=wobj_JMora;
        MoveL Target_3840,v60,z1,MarcadorVirtual\WObj:=wobj_JMora;
        MoveL Target_3850,v60,z1,MarcadorVirtual\WObj:=wobj_JMora;
        MoveL Target_3860,v60,z1,MarcadorVirtual\WObj:=wobj_JMora;
        MoveL Target_3870,v60,z1,MarcadorVirtual\WObj:=wobj_JMora;
        MoveL Target_3880,v60,z1,MarcadorVirtual\WObj:=wobj_JMora;
        MoveL Target_3890,v60,z1,MarcadorVirtual\WObj:=wobj_JMora;
        MoveL Target_3900,v60,z1,MarcadorVirtual\WObj:=wobj_JMora;
        MoveL Target_3910,v60,z1,MarcadorVirtual\WObj:=wobj_JMora;
        MoveL Target_3920,v60,z1,MarcadorVirtual\WObj:=wobj_JMora;
        MoveL Target_3930,v60,z1,MarcadorVirtual\WObj:=wobj_JMora;
        MoveL Target_3940,v60,z1,MarcadorVirtual\WObj:=wobj_JMora;
        MoveL Target_3950,v60,z1,MarcadorVirtual\WObj:=wobj_JMora;
        MoveL Target_3960,v60,z1,MarcadorVirtual\WObj:=wobj_JMora;
        MoveL Target_3970,v60,z1,MarcadorVirtual\WObj:=wobj_JMora;
        MoveL Target_3980,v60,z1,MarcadorVirtual\WObj:=wobj_JMora;
        MoveL Target_3990,v60,z1,MarcadorVirtual\WObj:=wobj_JMora;
        MoveL Target_4000,v60,z1,MarcadorVirtual\WObj:=wobj_JMora;
        MoveL Target_4010,v60,z1,MarcadorVirtual\WObj:=wobj_JMora;
        MoveL Target_4020,v60,z1,MarcadorVirtual\WObj:=wobj_JMora;
        MoveL Target_4030,v60,z1,MarcadorVirtual\WObj:=wobj_JMora;
        MoveL Target_4040,v60,z1,MarcadorVirtual\WObj:=wobj_JMora;
        MoveL Target_4050,v60,z1,MarcadorVirtual\WObj:=wobj_JMora;
        MoveL Target_4060,v60,z1,MarcadorVirtual\WObj:=wobj_JMora;
        MoveL Target_4070,v60,z1,MarcadorVirtual\WObj:=wobj_JMora;
        MoveL Target_4080,v60,z1,MarcadorVirtual\WObj:=wobj_JMora;
        MoveL Target_4090,v60,z1,MarcadorVirtual\WObj:=wobj_JMora;
        MoveL Target_4100,v60,z1,MarcadorVirtual\WObj:=wobj_JMora;
        MoveL Target_4110,v60,z1,MarcadorVirtual\WObj:=wobj_JMora;
        MoveL Target_4120,v60,z1,MarcadorVirtual\WObj:=wobj_JMora;
        MoveL Target_4130,v60,z1,MarcadorVirtual\WObj:=wobj_JMora;
        MoveL Target_4140,v60,z1,MarcadorVirtual\WObj:=wobj_JMora;
        MoveL Target_4150,v60,z1,MarcadorVirtual\WObj:=wobj_JMora;
        MoveL Target_4160,v60,z1,MarcadorVirtual\WObj:=wobj_JMora;
        MoveL Target_4170,v60,z1,MarcadorVirtual\WObj:=wobj_JMora;
        MoveL Target_4180,v60,z1,MarcadorVirtual\WObj:=wobj_JMora;
        MoveL Target_4190,v60,z1,MarcadorVirtual\WObj:=wobj_JMora;
        MoveL Target_4200,v60,z1,MarcadorVirtual\WObj:=wobj_JMora;
        MoveL Target_4210,v60,z1,MarcadorVirtual\WObj:=wobj_JMora;
        MoveL Target_4220,v60,z1,MarcadorVirtual\WObj:=wobj_JMora;
        MoveL Target_4230,v60,z1,MarcadorVirtual\WObj:=wobj_JMora;
        MoveL Target_4240,v60,z1,MarcadorVirtual\WObj:=wobj_JMora;
        MoveL Target_4250,v60,z1,MarcadorVirtual\WObj:=wobj_JMora;
    ENDPROC
    PROC Path_A2()
        MoveL Target_4260,v60,z1,MarcadorVirtual\WObj:=wobj_JMora;
        MoveL Target_4270,v60,z1,MarcadorVirtual\WObj:=wobj_JMora;
        MoveL Target_4280,v60,z1,MarcadorVirtual\WObj:=wobj_JMora;
        MoveL Target_4290,v60,z1,MarcadorVirtual\WObj:=wobj_JMora;
        MoveL Target_4300,v60,z1,MarcadorVirtual\WObj:=wobj_JMora;
        MoveL Target_4310,v60,z1,MarcadorVirtual\WObj:=wobj_JMora;
        MoveL Target_4320,v60,z1,MarcadorVirtual\WObj:=wobj_JMora;
        MoveL Target_4330,v60,z1,MarcadorVirtual\WObj:=wobj_JMora;
        MoveL Target_4340,v60,z1,MarcadorVirtual\WObj:=wobj_JMora;
        MoveL Target_4350,v60,z1,MarcadorVirtual\WObj:=wobj_JMora;
        MoveL Target_4360,v60,z1,MarcadorVirtual\WObj:=wobj_JMora;
        MoveL Target_4370,v60,z1,MarcadorVirtual\WObj:=wobj_JMora;
        MoveL Target_4380,v60,z1,MarcadorVirtual\WObj:=wobj_JMora;
        MoveL Target_4390,v60,z1,MarcadorVirtual\WObj:=wobj_JMora;
        MoveL Target_4400,v60,z1,MarcadorVirtual\WObj:=wobj_JMora;
        MoveL Target_4410,v60,z1,MarcadorVirtual\WObj:=wobj_JMora;
        MoveL Target_4420,v60,z1,MarcadorVirtual\WObj:=wobj_JMora;
        MoveL Target_4430,v60,z1,MarcadorVirtual\WObj:=wobj_JMora;
        MoveL Target_4440,v60,z1,MarcadorVirtual\WObj:=wobj_JMora;
        MoveL Target_4450,v60,z1,MarcadorVirtual\WObj:=wobj_JMora;
        MoveL Target_4460,v60,z1,MarcadorVirtual\WObj:=wobj_JMora;
        MoveL Target_4470,v60,z1,MarcadorVirtual\WObj:=wobj_JMora;
        MoveL Target_4480,v60,z1,MarcadorVirtual\WObj:=wobj_JMora;
        MoveL Target_4490,v60,z1,MarcadorVirtual\WObj:=wobj_JMora;
        MoveL Target_4500,v60,z1,MarcadorVirtual\WObj:=wobj_JMora;
        MoveL Target_4510,v60,z1,MarcadorVirtual\WObj:=wobj_JMora;
        MoveL Target_4520,v60,z1,MarcadorVirtual\WObj:=wobj_JMora;
        MoveL Target_4530,v60,z1,MarcadorVirtual\WObj:=wobj_JMora;
        MoveL Target_4540,v60,z1,MarcadorVirtual\WObj:=wobj_JMora;
        MoveL Target_4550,v60,z1,MarcadorVirtual\WObj:=wobj_JMora;
        MoveL Target_4560,v60,z1,MarcadorVirtual\WObj:=wobj_JMora;
        MoveL Target_4570,v60,z1,MarcadorVirtual\WObj:=wobj_JMora;
        MoveL Target_4580,v60,z1,MarcadorVirtual\WObj:=wobj_JMora;
        MoveL Target_4590,v60,z1,MarcadorVirtual\WObj:=wobj_JMora;
        MoveL Target_4600,v60,z1,MarcadorVirtual\WObj:=wobj_JMora;
        MoveL Target_4610,v60,z1,MarcadorVirtual\WObj:=wobj_JMora;
        MoveL Target_4620,v60,z1,MarcadorVirtual\WObj:=wobj_JMora;
        MoveL Target_4630,v60,z1,MarcadorVirtual\WObj:=wobj_JMora;
        MoveL Target_4640,v60,z1,MarcadorVirtual\WObj:=wobj_JMora;
        MoveL Target_4650,v60,z1,MarcadorVirtual\WObj:=wobj_JMora;
        MoveL Target_4660,v60,z1,MarcadorVirtual\WObj:=wobj_JMora;
        MoveL Target_4670,v60,z1,MarcadorVirtual\WObj:=wobj_JMora;
        MoveL Target_4680,v60,z1,MarcadorVirtual\WObj:=wobj_JMora;
        MoveL Target_4690,v60,z1,MarcadorVirtual\WObj:=wobj_JMora;
        MoveL Target_4700,v60,z1,MarcadorVirtual\WObj:=wobj_JMora;
        MoveL Target_4710,v60,z1,MarcadorVirtual\WObj:=wobj_JMora;
        MoveL Target_4720,v60,z1,MarcadorVirtual\WObj:=wobj_JMora;
        MoveL Target_4730,v60,z1,MarcadorVirtual\WObj:=wobj_JMora;
        MoveL Target_4740,v60,z1,MarcadorVirtual\WObj:=wobj_JMora;
        MoveL Target_4750,v60,z1,MarcadorVirtual\WObj:=wobj_JMora;
        MoveL Target_4760,v60,z1,MarcadorVirtual\WObj:=wobj_JMora;
        MoveL Target_4770,v60,z1,MarcadorVirtual\WObj:=wobj_JMora;
        MoveL Target_4780,v60,z1,MarcadorVirtual\WObj:=wobj_JMora;
        MoveL Target_4790,v60,z1,MarcadorVirtual\WObj:=wobj_JMora;
        MoveL Target_4800,v60,z1,MarcadorVirtual\WObj:=wobj_JMora;
        MoveL Target_4810,v60,z1,MarcadorVirtual\WObj:=wobj_JMora;
        MoveL Target_4820,v60,z1,MarcadorVirtual\WObj:=wobj_JMora;
        MoveL Target_4830,v60,z1,MarcadorVirtual\WObj:=wobj_JMora;
        MoveL Target_4840,v60,z1,MarcadorVirtual\WObj:=wobj_JMora;
        MoveL Target_4850,v60,z1,MarcadorVirtual\WObj:=wobj_JMora;
        MoveL Target_4860,v60,z1,MarcadorVirtual\WObj:=wobj_JMora;
        MoveL Target_4870,v60,z1,MarcadorVirtual\WObj:=wobj_JMora;
        MoveL Target_4880,v60,z1,MarcadorVirtual\WObj:=wobj_JMora;
        MoveL Target_4890,v60,z1,MarcadorVirtual\WObj:=wobj_JMora;
        MoveL Target_4900,v60,z1,MarcadorVirtual\WObj:=wobj_JMora;
        MoveL Target_4910,v60,z1,MarcadorVirtual\WObj:=wobj_JMora;
        MoveL Target_4920,v60,z1,MarcadorVirtual\WObj:=wobj_JMora;
        MoveL Target_4930,v60,z1,MarcadorVirtual\WObj:=wobj_JMora;
        MoveL Target_4940,v60,z1,MarcadorVirtual\WObj:=wobj_JMora;
        MoveL Target_4950,v60,z1,MarcadorVirtual\WObj:=wobj_JMora;
        MoveL Target_4960,v60,z1,MarcadorVirtual\WObj:=wobj_JMora;
        MoveL Target_4970,v60,z1,MarcadorVirtual\WObj:=wobj_JMora;
        MoveL Target_4980,v60,z1,MarcadorVirtual\WObj:=wobj_JMora;
        MoveL Target_4990,v60,z1,MarcadorVirtual\WObj:=wobj_JMora;
        MoveL Target_5000,v60,z1,MarcadorVirtual\WObj:=wobj_JMora;
        MoveL Target_5010,v60,z1,MarcadorVirtual\WObj:=wobj_JMora;
        MoveL Target_5020,v60,z1,MarcadorVirtual\WObj:=wobj_JMora;
        MoveL Target_5030,v60,z1,MarcadorVirtual\WObj:=wobj_JMora;
        MoveL Target_5040,v60,z1,MarcadorVirtual\WObj:=wobj_JMora;
        MoveL Target_5050,v60,z1,MarcadorVirtual\WObj:=wobj_JMora;
    ENDPROC
    PROC Path_G()
        MoveL Target_5060,v60,z1,MarcadorVirtual\WObj:=wobj_JMora;
        MoveL Target_5070,v60,z1,MarcadorVirtual\WObj:=wobj_JMora;
        MoveL Target_5080,v60,z1,MarcadorVirtual\WObj:=wobj_JMora;
        MoveL Target_5090,v60,z1,MarcadorVirtual\WObj:=wobj_JMora;
        MoveL Target_5100,v60,z1,MarcadorVirtual\WObj:=wobj_JMora;
        MoveL Target_5110,v60,z1,MarcadorVirtual\WObj:=wobj_JMora;
        MoveL Target_5120,v60,z1,MarcadorVirtual\WObj:=wobj_JMora;
        MoveL Target_5130,v60,z1,MarcadorVirtual\WObj:=wobj_JMora;
        MoveL Target_5140,v60,z1,MarcadorVirtual\WObj:=wobj_JMora;
        MoveL Target_5150,v60,z1,MarcadorVirtual\WObj:=wobj_JMora;
        MoveL Target_5160,v60,z1,MarcadorVirtual\WObj:=wobj_JMora;
        MoveL Target_5170,v60,z1,MarcadorVirtual\WObj:=wobj_JMora;
        MoveL Target_5180,v60,z1,MarcadorVirtual\WObj:=wobj_JMora;
        MoveL Target_5190,v60,z1,MarcadorVirtual\WObj:=wobj_JMora;
        MoveL Target_5200,v60,z1,MarcadorVirtual\WObj:=wobj_JMora;
        MoveL Target_5210,v60,z1,MarcadorVirtual\WObj:=wobj_JMora;
        MoveL Target_5220,v60,z1,MarcadorVirtual\WObj:=wobj_JMora;
        MoveL Target_5230,v60,z1,MarcadorVirtual\WObj:=wobj_JMora;
        MoveL Target_5240,v60,z1,MarcadorVirtual\WObj:=wobj_JMora;
        MoveL Target_5250,v60,z1,MarcadorVirtual\WObj:=wobj_JMora;
        MoveL Target_5260,v60,z1,MarcadorVirtual\WObj:=wobj_JMora;
        MoveL Target_5270,v60,z1,MarcadorVirtual\WObj:=wobj_JMora;
        MoveL Target_5280,v60,z1,MarcadorVirtual\WObj:=wobj_JMora;
        MoveL Target_5290,v60,z1,MarcadorVirtual\WObj:=wobj_JMora;
        MoveL Target_5300,v60,z1,MarcadorVirtual\WObj:=wobj_JMora;
        MoveL Target_5310,v60,z1,MarcadorVirtual\WObj:=wobj_JMora;
        MoveL Target_5320,v60,z1,MarcadorVirtual\WObj:=wobj_JMora;
        MoveL Target_5330,v60,z1,MarcadorVirtual\WObj:=wobj_JMora;
        MoveL Target_5340,v60,z1,MarcadorVirtual\WObj:=wobj_JMora;
        MoveL Target_5350,v60,z1,MarcadorVirtual\WObj:=wobj_JMora;
        MoveL Target_5360,v60,z1,MarcadorVirtual\WObj:=wobj_JMora;
        MoveL Target_5370,v60,z1,MarcadorVirtual\WObj:=wobj_JMora;
        MoveL Target_5380,v60,z1,MarcadorVirtual\WObj:=wobj_JMora;
        MoveL Target_5390,v60,z1,MarcadorVirtual\WObj:=wobj_JMora;
        MoveL Target_5400,v60,z1,MarcadorVirtual\WObj:=wobj_JMora;
        MoveL Target_5410,v60,z1,MarcadorVirtual\WObj:=wobj_JMora;
        MoveL Target_5420,v60,z1,MarcadorVirtual\WObj:=wobj_JMora;
        MoveL Target_5430,v60,z1,MarcadorVirtual\WObj:=wobj_JMora;
        MoveL Target_5440,v60,z1,MarcadorVirtual\WObj:=wobj_JMora;
        MoveL Target_5450,v60,z1,MarcadorVirtual\WObj:=wobj_JMora;
        MoveL Target_5460,v60,z1,MarcadorVirtual\WObj:=wobj_JMora;
        MoveL Target_5470,v60,z1,MarcadorVirtual\WObj:=wobj_JMora;
        MoveL Target_5480,v60,z1,MarcadorVirtual\WObj:=wobj_JMora;
        MoveL Target_5490,v60,z1,MarcadorVirtual\WObj:=wobj_JMora;
        MoveL Target_5500,v60,z1,MarcadorVirtual\WObj:=wobj_JMora;
        MoveL Target_5510,v60,z1,MarcadorVirtual\WObj:=wobj_JMora;
        MoveL Target_5520,v60,z1,MarcadorVirtual\WObj:=wobj_JMora;
        MoveL Target_5530,v60,z1,MarcadorVirtual\WObj:=wobj_JMora;
        MoveL Target_5540,v60,z1,MarcadorVirtual\WObj:=wobj_JMora;
        MoveL Target_5550,v60,z1,MarcadorVirtual\WObj:=wobj_JMora;
        MoveL Target_5560,v60,z1,MarcadorVirtual\WObj:=wobj_JMora;
        MoveL Target_5570,v60,z1,MarcadorVirtual\WObj:=wobj_JMora;
        MoveL Target_5580,v60,z1,MarcadorVirtual\WObj:=wobj_JMora;
        MoveL Target_5590,v60,z1,MarcadorVirtual\WObj:=wobj_JMora;
        MoveL Target_5600,v60,z1,MarcadorVirtual\WObj:=wobj_JMora;
        MoveL Target_5610,v60,z1,MarcadorVirtual\WObj:=wobj_JMora;
        MoveL Target_5620,v60,z1,MarcadorVirtual\WObj:=wobj_JMora;
        MoveL Target_5630,v60,z1,MarcadorVirtual\WObj:=wobj_JMora;
        MoveL Target_5640,v60,z1,MarcadorVirtual\WObj:=wobj_JMora;
        MoveL Target_5650,v60,z1,MarcadorVirtual\WObj:=wobj_JMora;
        MoveL Target_5660,v60,z1,MarcadorVirtual\WObj:=wobj_JMora;
        MoveL Target_5670,v60,z1,MarcadorVirtual\WObj:=wobj_JMora;
        MoveL Target_5680,v60,z1,MarcadorVirtual\WObj:=wobj_JMora;
        MoveL Target_5690,v60,z1,MarcadorVirtual\WObj:=wobj_JMora;
        MoveL Target_5700,v60,z1,MarcadorVirtual\WObj:=wobj_JMora;
        MoveL Target_5710,v60,z1,MarcadorVirtual\WObj:=wobj_JMora;
        MoveL Target_5720,v60,z1,MarcadorVirtual\WObj:=wobj_JMora;
        MoveL Target_5730,v60,z1,MarcadorVirtual\WObj:=wobj_JMora;
        MoveL Target_5740,v60,z1,MarcadorVirtual\WObj:=wobj_JMora;
        MoveL Target_5750,v60,z1,MarcadorVirtual\WObj:=wobj_JMora;
        MoveL Target_5760,v60,z1,MarcadorVirtual\WObj:=wobj_JMora;
        MoveL Target_5770,v60,z1,MarcadorVirtual\WObj:=wobj_JMora;
        MoveL Target_5780,v60,z1,MarcadorVirtual\WObj:=wobj_JMora;
        MoveL Target_5790,v60,z1,MarcadorVirtual\WObj:=wobj_JMora;
        MoveL Target_5800,v60,z1,MarcadorVirtual\WObj:=wobj_JMora;
        MoveL Target_5810,v60,z1,MarcadorVirtual\WObj:=wobj_JMora;
        MoveL Target_5820,v60,z1,MarcadorVirtual\WObj:=wobj_JMora;
        MoveL Target_5830,v60,z1,MarcadorVirtual\WObj:=wobj_JMora;
        MoveL Target_5840,v60,z1,MarcadorVirtual\WObj:=wobj_JMora;
        MoveL Target_5850,v60,z1,MarcadorVirtual\WObj:=wobj_JMora;
        MoveL Target_5860,v60,z1,MarcadorVirtual\WObj:=wobj_JMora;
        MoveL Target_5870,v60,z1,MarcadorVirtual\WObj:=wobj_JMora;
        MoveL Target_5880,v60,z1,MarcadorVirtual\WObj:=wobj_JMora;
        MoveL Target_5890,v60,z1,MarcadorVirtual\WObj:=wobj_JMora;
        MoveL Target_5900,v60,z1,MarcadorVirtual\WObj:=wobj_JMora;
        MoveL Target_5910,v60,z1,MarcadorVirtual\WObj:=wobj_JMora;
        MoveL Target_5920,v60,z1,MarcadorVirtual\WObj:=wobj_JMora;
        MoveL Target_5930,v60,z1,MarcadorVirtual\WObj:=wobj_JMora;
    ENDPROC
    PROC Path_U2()
        MoveL Target_5940,v60,z1,MarcadorVirtual\WObj:=wobj_JMora;
        MoveL Target_5950,v60,z1,MarcadorVirtual\WObj:=wobj_JMora;
        MoveL Target_5960,v60,z1,MarcadorVirtual\WObj:=wobj_JMora;
        MoveL Target_5970,v60,z1,MarcadorVirtual\WObj:=wobj_JMora;
        MoveL Target_5980,v60,z1,MarcadorVirtual\WObj:=wobj_JMora;
        MoveL Target_5990,v60,z1,MarcadorVirtual\WObj:=wobj_JMora;
        MoveL Target_6000,v60,z1,MarcadorVirtual\WObj:=wobj_JMora;
        MoveL Target_6010,v60,z1,MarcadorVirtual\WObj:=wobj_JMora;
        MoveL Target_6020,v60,z1,MarcadorVirtual\WObj:=wobj_JMora;
        MoveL Target_6030,v60,z1,MarcadorVirtual\WObj:=wobj_JMora;
        MoveL Target_6040,v60,z1,MarcadorVirtual\WObj:=wobj_JMora;
        MoveL Target_6050,v60,z1,MarcadorVirtual\WObj:=wobj_JMora;
        MoveL Target_6060,v60,z1,MarcadorVirtual\WObj:=wobj_JMora;
        MoveL Target_6070,v60,z1,MarcadorVirtual\WObj:=wobj_JMora;
        MoveL Target_6080,v60,z1,MarcadorVirtual\WObj:=wobj_JMora;
        MoveL Target_6090,v60,z1,MarcadorVirtual\WObj:=wobj_JMora;
        MoveL Target_6100,v60,z1,MarcadorVirtual\WObj:=wobj_JMora;
        MoveL Target_6110,v60,z1,MarcadorVirtual\WObj:=wobj_JMora;
        MoveL Target_6120,v60,z1,MarcadorVirtual\WObj:=wobj_JMora;
        MoveL Target_6130,v60,z1,MarcadorVirtual\WObj:=wobj_JMora;
        MoveL Target_6140,v60,z1,MarcadorVirtual\WObj:=wobj_JMora;
        MoveL Target_6150,v60,z1,MarcadorVirtual\WObj:=wobj_JMora;
        MoveL Target_6160,v60,z1,MarcadorVirtual\WObj:=wobj_JMora;
        MoveL Target_6170,v60,z1,MarcadorVirtual\WObj:=wobj_JMora;
        MoveL Target_6180,v60,z1,MarcadorVirtual\WObj:=wobj_JMora;
        MoveL Target_6190,v60,z1,MarcadorVirtual\WObj:=wobj_JMora;
        MoveL Target_6200,v60,z1,MarcadorVirtual\WObj:=wobj_JMora;
        MoveL Target_6210,v60,z1,MarcadorVirtual\WObj:=wobj_JMora;
        MoveL Target_6220,v60,z1,MarcadorVirtual\WObj:=wobj_JMora;
        MoveL Target_6230,v60,z1,MarcadorVirtual\WObj:=wobj_JMora;
        MoveL Target_6240,v60,z1,MarcadorVirtual\WObj:=wobj_JMora;
        MoveL Target_6250,v60,z1,MarcadorVirtual\WObj:=wobj_JMora;
        MoveL Target_6260,v60,z1,MarcadorVirtual\WObj:=wobj_JMora;
        MoveL Target_6270,v60,z1,MarcadorVirtual\WObj:=wobj_JMora;
        MoveL Target_6280,v60,z1,MarcadorVirtual\WObj:=wobj_JMora;
        MoveL Target_6290,v60,z1,MarcadorVirtual\WObj:=wobj_JMora;
        MoveL Target_6300,v60,z1,MarcadorVirtual\WObj:=wobj_JMora;
        MoveL Target_6310,v60,z1,MarcadorVirtual\WObj:=wobj_JMora;
        MoveL Target_6320,v60,z1,MarcadorVirtual\WObj:=wobj_JMora;
        MoveL Target_6330,v60,z1,MarcadorVirtual\WObj:=wobj_JMora;
        MoveL Target_6340,v60,z1,MarcadorVirtual\WObj:=wobj_JMora;
        MoveL Target_6350,v60,z1,MarcadorVirtual\WObj:=wobj_JMora;
        MoveL Target_6360,v60,z1,MarcadorVirtual\WObj:=wobj_JMora;
        MoveL Target_6370,v60,z1,MarcadorVirtual\WObj:=wobj_JMora;
        MoveL Target_6380,v60,z1,MarcadorVirtual\WObj:=wobj_JMora;
        MoveL Target_6390,v60,z1,MarcadorVirtual\WObj:=wobj_JMora;
    ENDPROC
    PROC Path_S()
        MoveL Target_6400,v60,z1,MarcadorVirtual\WObj:=wobj_JMora;
        MoveL Target_6410,v60,z1,MarcadorVirtual\WObj:=wobj_JMora;
        MoveL Target_6420,v60,z1,MarcadorVirtual\WObj:=wobj_JMora;
        MoveL Target_6430,v60,z1,MarcadorVirtual\WObj:=wobj_JMora;
        MoveL Target_6440,v60,z1,MarcadorVirtual\WObj:=wobj_JMora;
        MoveL Target_6450,v60,z1,MarcadorVirtual\WObj:=wobj_JMora;
        MoveL Target_6460,v60,z1,MarcadorVirtual\WObj:=wobj_JMora;
        MoveL Target_6470,v60,z1,MarcadorVirtual\WObj:=wobj_JMora;
        MoveL Target_6480,v60,z1,MarcadorVirtual\WObj:=wobj_JMora;
        MoveL Target_6490,v60,z1,MarcadorVirtual\WObj:=wobj_JMora;
        MoveL Target_6500,v60,z1,MarcadorVirtual\WObj:=wobj_JMora;
        MoveL Target_6510,v60,z1,MarcadorVirtual\WObj:=wobj_JMora;
        MoveL Target_6520,v60,z1,MarcadorVirtual\WObj:=wobj_JMora;
        MoveL Target_6530,v60,z1,MarcadorVirtual\WObj:=wobj_JMora;
        MoveL Target_6540,v60,z1,MarcadorVirtual\WObj:=wobj_JMora;
        MoveL Target_6550,v60,z1,MarcadorVirtual\WObj:=wobj_JMora;
        MoveL Target_6560,v60,z1,MarcadorVirtual\WObj:=wobj_JMora;
        MoveL Target_6570,v60,z1,MarcadorVirtual\WObj:=wobj_JMora;
        MoveL Target_6580,v60,z1,MarcadorVirtual\WObj:=wobj_JMora;
        MoveL Target_6590,v60,z1,MarcadorVirtual\WObj:=wobj_JMora;
        MoveL Target_6600,v60,z1,MarcadorVirtual\WObj:=wobj_JMora;
        MoveL Target_6610,v60,z1,MarcadorVirtual\WObj:=wobj_JMora;
        MoveL Target_6620,v60,z1,MarcadorVirtual\WObj:=wobj_JMora;
        MoveL Target_6630,v60,z1,MarcadorVirtual\WObj:=wobj_JMora;
        MoveL Target_6640,v60,z1,MarcadorVirtual\WObj:=wobj_JMora;
        MoveL Target_6650,v60,z1,MarcadorVirtual\WObj:=wobj_JMora;
        MoveL Target_6660,v60,z1,MarcadorVirtual\WObj:=wobj_JMora;
        MoveL Target_6670,v60,z1,MarcadorVirtual\WObj:=wobj_JMora;
        MoveL Target_6680,v60,z1,MarcadorVirtual\WObj:=wobj_JMora;
        MoveL Target_6690,v60,z1,MarcadorVirtual\WObj:=wobj_JMora;
        MoveL Target_6700,v60,z1,MarcadorVirtual\WObj:=wobj_JMora;
        MoveL Target_6710,v60,z1,MarcadorVirtual\WObj:=wobj_JMora;
        MoveL Target_6720,v60,z1,MarcadorVirtual\WObj:=wobj_JMora;
        MoveL Target_6730,v60,z1,MarcadorVirtual\WObj:=wobj_JMora;
        MoveL Target_6740,v60,z1,MarcadorVirtual\WObj:=wobj_JMora;
        MoveL Target_6750,v60,z1,MarcadorVirtual\WObj:=wobj_JMora;
        MoveL Target_6760,v60,z1,MarcadorVirtual\WObj:=wobj_JMora;
        MoveL Target_6770,v60,z1,MarcadorVirtual\WObj:=wobj_JMora;
        MoveL Target_6780,v60,z1,MarcadorVirtual\WObj:=wobj_JMora;
        MoveL Target_6790,v60,z1,MarcadorVirtual\WObj:=wobj_JMora;
        MoveL Target_6800,v60,z1,MarcadorVirtual\WObj:=wobj_JMora;
        MoveL Target_6810,v60,z1,MarcadorVirtual\WObj:=wobj_JMora;
        MoveL Target_6820,v60,z1,MarcadorVirtual\WObj:=wobj_JMora;
        MoveL Target_6830,v60,z1,MarcadorVirtual\WObj:=wobj_JMora;
        MoveL Target_6840,v60,z1,MarcadorVirtual\WObj:=wobj_JMora;
        MoveL Target_6850,v60,z1,MarcadorVirtual\WObj:=wobj_JMora;
        MoveL Target_6860,v60,z1,MarcadorVirtual\WObj:=wobj_JMora;
        MoveL Target_6870,v60,z1,MarcadorVirtual\WObj:=wobj_JMora;
        MoveL Target_6880,v60,z1,MarcadorVirtual\WObj:=wobj_JMora;
        MoveL Target_6890,v60,z1,MarcadorVirtual\WObj:=wobj_JMora;
        MoveL Target_6900,v60,z1,MarcadorVirtual\WObj:=wobj_JMora;
        MoveL Target_6910,v60,z1,MarcadorVirtual\WObj:=wobj_JMora;
        MoveL Target_6920,v60,z1,MarcadorVirtual\WObj:=wobj_JMora;
        MoveL Target_6930,v60,z1,MarcadorVirtual\WObj:=wobj_JMora;
        MoveL Target_6940,v60,z1,MarcadorVirtual\WObj:=wobj_JMora;
        MoveL Target_6950,v60,z1,MarcadorVirtual\WObj:=wobj_JMora;
        MoveL Target_6960,v60,z1,MarcadorVirtual\WObj:=wobj_JMora;
        MoveL Target_6970,v60,z1,MarcadorVirtual\WObj:=wobj_JMora;
        MoveL Target_6980,v60,z1,MarcadorVirtual\WObj:=wobj_JMora;
        MoveL Target_6990,v60,z1,MarcadorVirtual\WObj:=wobj_JMora;
        MoveL Target_7000,v60,z1,MarcadorVirtual\WObj:=wobj_JMora;
        MoveL Target_7010,v60,z1,MarcadorVirtual\WObj:=wobj_JMora;
        MoveL Target_7020,v60,z1,MarcadorVirtual\WObj:=wobj_JMora;
        MoveL Target_7030,v60,z1,MarcadorVirtual\WObj:=wobj_JMora;
        MoveL Target_7040,v60,z1,MarcadorVirtual\WObj:=wobj_JMora;
        MoveL Target_7050,v60,z1,MarcadorVirtual\WObj:=wobj_JMora;
        MoveL Target_7060,v60,z1,MarcadorVirtual\WObj:=wobj_JMora;
        MoveL Target_7070,v60,z1,MarcadorVirtual\WObj:=wobj_JMora;
        MoveL Target_7080,v60,z1,MarcadorVirtual\WObj:=wobj_JMora;
        MoveL Target_7090,v60,z1,MarcadorVirtual\WObj:=wobj_JMora;
        MoveL Target_7100,v60,z1,MarcadorVirtual\WObj:=wobj_JMora;
        MoveL Target_7110,v60,z1,MarcadorVirtual\WObj:=wobj_JMora;
        MoveL Target_7120,v60,z1,MarcadorVirtual\WObj:=wobj_JMora;
        MoveL Target_7130,v60,z1,MarcadorVirtual\WObj:=wobj_JMora;
        MoveL Target_7140,v60,z1,MarcadorVirtual\WObj:=wobj_JMora;
        MoveL Target_7150,v60,z1,MarcadorVirtual\WObj:=wobj_JMora;
        MoveL Target_7160,v60,z1,MarcadorVirtual\WObj:=wobj_JMora;
        MoveL Target_7170,v60,z1,MarcadorVirtual\WObj:=wobj_JMora;
        MoveL Target_7180,v60,z1,MarcadorVirtual\WObj:=wobj_JMora;
        MoveL Target_7190,v60,z1,MarcadorVirtual\WObj:=wobj_JMora;
        MoveL Target_7200,v60,z1,MarcadorVirtual\WObj:=wobj_JMora;
        MoveL Target_7210,v60,z1,MarcadorVirtual\WObj:=wobj_JMora;
        MoveL Target_7220,v60,z1,MarcadorVirtual\WObj:=wobj_JMora;
        MoveL Target_7230,v60,z1,MarcadorVirtual\WObj:=wobj_JMora;
        MoveL Target_7240,v60,z1,MarcadorVirtual\WObj:=wobj_JMora;
        MoveL Target_7250,v60,z1,MarcadorVirtual\WObj:=wobj_JMora;
        MoveL Target_7260,v60,z1,MarcadorVirtual\WObj:=wobj_JMora;
        MoveL Target_7270,v60,z1,MarcadorVirtual\WObj:=wobj_JMora;
        MoveL Target_7280,v60,z1,MarcadorVirtual\WObj:=wobj_JMora;
        MoveL Target_7290,v60,z1,MarcadorVirtual\WObj:=wobj_JMora;
        MoveL Target_7300,v60,z1,MarcadorVirtual\WObj:=wobj_JMora;
        MoveL Target_7310,v60,z1,MarcadorVirtual\WObj:=wobj_JMora;
        MoveL Target_7320,v60,z1,MarcadorVirtual\WObj:=wobj_JMora;
        MoveL Target_7330,v60,z1,MarcadorVirtual\WObj:=wobj_JMora;
    ENDPROC
    PROC Path_T()
        MoveL Target_7340,v60,z1,MarcadorVirtual\WObj:=wobj_JMora;
        MoveL Target_7350,v60,z1,MarcadorVirtual\WObj:=wobj_JMora;
        MoveL Target_7360,v60,z1,MarcadorVirtual\WObj:=wobj_JMora;
        MoveL Target_7370,v60,z1,MarcadorVirtual\WObj:=wobj_JMora;
        MoveL Target_7380,v60,z1,MarcadorVirtual\WObj:=wobj_JMora;
        MoveL Target_7390,v60,z1,MarcadorVirtual\WObj:=wobj_JMora;
        MoveL Target_7400,v60,z1,MarcadorVirtual\WObj:=wobj_JMora;
        MoveL Target_7410,v60,z1,MarcadorVirtual\WObj:=wobj_JMora;
        MoveL Target_7420,v60,z1,MarcadorVirtual\WObj:=wobj_JMora;
        MoveL Target_7430,v60,z1,MarcadorVirtual\WObj:=wobj_JMora;
        MoveL Target_7440,v60,z1,MarcadorVirtual\WObj:=wobj_JMora;
        MoveL Target_7450,v60,z1,MarcadorVirtual\WObj:=wobj_JMora;
        MoveL Target_7460,v60,z1,MarcadorVirtual\WObj:=wobj_JMora;
        MoveL Target_7470,v60,z1,MarcadorVirtual\WObj:=wobj_JMora;
        MoveL Target_7480,v60,z1,MarcadorVirtual\WObj:=wobj_JMora;
        MoveL Target_7490,v60,z1,MarcadorVirtual\WObj:=wobj_JMora;
        MoveL Target_7500,v60,z1,MarcadorVirtual\WObj:=wobj_JMora;
        MoveL Target_7510,v60,z1,MarcadorVirtual\WObj:=wobj_JMora;
        MoveL Target_7520,v60,z1,MarcadorVirtual\WObj:=wobj_JMora;
        MoveL Target_7530,v60,z1,MarcadorVirtual\WObj:=wobj_JMora;
        MoveL Target_7540,v60,z1,MarcadorVirtual\WObj:=wobj_JMora;
        MoveL Target_7550,v60,z1,MarcadorVirtual\WObj:=wobj_JMora;
        MoveL Target_7560,v60,z1,MarcadorVirtual\WObj:=wobj_JMora;
        MoveL Target_7570,v60,z1,MarcadorVirtual\WObj:=wobj_JMora;
        MoveL Target_7580,v60,z1,MarcadorVirtual\WObj:=wobj_JMora;
        MoveL Target_7590,v60,z1,MarcadorVirtual\WObj:=wobj_JMora;
        MoveL Target_7600,v60,z1,MarcadorVirtual\WObj:=wobj_JMora;
        MoveL Target_7610,v60,z1,MarcadorVirtual\WObj:=wobj_JMora;
        MoveL Target_7620,v60,z1,MarcadorVirtual\WObj:=wobj_JMora;
        MoveL Target_7630,v60,z1,MarcadorVirtual\WObj:=wobj_JMora;
        MoveL Target_7640,v60,z1,MarcadorVirtual\WObj:=wobj_JMora;
        MoveL Target_7650,v60,z1,MarcadorVirtual\WObj:=wobj_JMora;
        MoveL Target_7660,v60,z1,MarcadorVirtual\WObj:=wobj_JMora;
        MoveL Target_7670,v60,z1,MarcadorVirtual\WObj:=wobj_JMora;
        MoveL Target_7680,v60,z1,MarcadorVirtual\WObj:=wobj_JMora;
        MoveL Target_7690,v60,z1,MarcadorVirtual\WObj:=wobj_JMora;
        MoveL Target_7700,v60,z1,MarcadorVirtual\WObj:=wobj_JMora;
        MoveL Target_7710,v60,z1,MarcadorVirtual\WObj:=wobj_JMora;
        MoveL Target_7720,v60,z1,MarcadorVirtual\WObj:=wobj_JMora;
        MoveL Target_7730,v60,z1,MarcadorVirtual\WObj:=wobj_JMora;
        MoveL Target_7740,v60,z1,MarcadorVirtual\WObj:=wobj_JMora;
        MoveL Target_7750,v60,z1,MarcadorVirtual\WObj:=wobj_JMora;
        MoveL Target_7760,v60,z1,MarcadorVirtual\WObj:=wobj_JMora;
        MoveL Target_7770,v60,z1,MarcadorVirtual\WObj:=wobj_JMora;
        MoveL Target_7780,v60,z1,MarcadorVirtual\WObj:=wobj_JMora;
        MoveL Target_7790,v60,z1,MarcadorVirtual\WObj:=wobj_JMora;
        MoveL Target_7800,v60,z1,MarcadorVirtual\WObj:=wobj_JMora;
        MoveL Target_7810,v60,z1,MarcadorVirtual\WObj:=wobj_JMora;
        MoveL Target_7820,v60,z1,MarcadorVirtual\WObj:=wobj_JMora;
        MoveL Target_7830,v60,z1,MarcadorVirtual\WObj:=wobj_JMora;
        MoveL Target_7840,v60,z1,MarcadorVirtual\WObj:=wobj_JMora;
        MoveL Target_7850,v60,z1,MarcadorVirtual\WObj:=wobj_JMora;
        MoveL Target_7860,v60,z1,MarcadorVirtual\WObj:=wobj_JMora;
        MoveL Target_7870,v60,z1,MarcadorVirtual\WObj:=wobj_JMora;
        MoveL Target_7880,v60,z1,MarcadorVirtual\WObj:=wobj_JMora;
        MoveL Target_7890,v60,z1,MarcadorVirtual\WObj:=wobj_JMora;
        MoveL Target_7900,v60,z1,MarcadorVirtual\WObj:=wobj_JMora;
        MoveL Target_7910,v60,z1,MarcadorVirtual\WObj:=wobj_JMora;
        MoveL Target_7920,v60,z1,MarcadorVirtual\WObj:=wobj_JMora;
        MoveL Target_7930,v60,z1,MarcadorVirtual\WObj:=wobj_JMora;
        MoveL Target_7940,v60,z1,MarcadorVirtual\WObj:=wobj_JMora;
        MoveL Target_7950,v60,z1,MarcadorVirtual\WObj:=wobj_JMora;
        MoveL Target_7960,v60,z1,MarcadorVirtual\WObj:=wobj_JMora;
        MoveL Target_7970,v60,z1,MarcadorVirtual\WObj:=wobj_JMora;
        MoveL Target_7980,v60,z1,MarcadorVirtual\WObj:=wobj_JMora;
        MoveL Target_7990,v60,z1,MarcadorVirtual\WObj:=wobj_JMora;
        MoveL Target_8000,v60,z1,MarcadorVirtual\WObj:=wobj_JMora;
    ENDPROC
    PROC Path_A3()
        MoveL Target_8010,v60,z1,MarcadorVirtual\WObj:=wobj_JMora;
        MoveL Target_8020,v60,z1,MarcadorVirtual\WObj:=wobj_JMora;
        MoveL Target_8030,v60,z1,MarcadorVirtual\WObj:=wobj_JMora;
        MoveL Target_8040,v60,z1,MarcadorVirtual\WObj:=wobj_JMora;
        MoveL Target_8050,v60,z1,MarcadorVirtual\WObj:=wobj_JMora;
        MoveL Target_8060,v60,z1,MarcadorVirtual\WObj:=wobj_JMora;
        MoveL Target_8070,v60,z1,MarcadorVirtual\WObj:=wobj_JMora;
        MoveL Target_8080,v60,z1,MarcadorVirtual\WObj:=wobj_JMora;
        MoveL Target_8090,v60,z1,MarcadorVirtual\WObj:=wobj_JMora;
        MoveL Target_8100,v60,z1,MarcadorVirtual\WObj:=wobj_JMora;
        MoveL Target_8110,v60,z1,MarcadorVirtual\WObj:=wobj_JMora;
        MoveL Target_8120,v60,z1,MarcadorVirtual\WObj:=wobj_JMora;
        MoveL Target_8130,v60,z1,MarcadorVirtual\WObj:=wobj_JMora;
        MoveL Target_8140,v60,z1,MarcadorVirtual\WObj:=wobj_JMora;
        MoveL Target_8150,v60,z1,MarcadorVirtual\WObj:=wobj_JMora;
        MoveL Target_8160,v60,z1,MarcadorVirtual\WObj:=wobj_JMora;
        MoveL Target_8170,v60,z1,MarcadorVirtual\WObj:=wobj_JMora;
        MoveL Target_8180,v60,z1,MarcadorVirtual\WObj:=wobj_JMora;
        MoveL Target_8190,v60,z1,MarcadorVirtual\WObj:=wobj_JMora;
        MoveL Target_8200,v60,z1,MarcadorVirtual\WObj:=wobj_JMora;
        MoveL Target_8210,v60,z1,MarcadorVirtual\WObj:=wobj_JMora;
        MoveL Target_8220,v60,z1,MarcadorVirtual\WObj:=wobj_JMora;
        MoveL Target_8230,v60,z1,MarcadorVirtual\WObj:=wobj_JMora;
        MoveL Target_8240,v60,z1,MarcadorVirtual\WObj:=wobj_JMora;
        MoveL Target_8250,v60,z1,MarcadorVirtual\WObj:=wobj_JMora;
        MoveL Target_8260,v60,z1,MarcadorVirtual\WObj:=wobj_JMora;
        MoveL Target_8270,v60,z1,MarcadorVirtual\WObj:=wobj_JMora;
        MoveL Target_8280,v60,z1,MarcadorVirtual\WObj:=wobj_JMora;
        MoveL Target_8290,v60,z1,MarcadorVirtual\WObj:=wobj_JMora;
        MoveL Target_8300,v60,z1,MarcadorVirtual\WObj:=wobj_JMora;
        MoveL Target_8310,v60,z1,MarcadorVirtual\WObj:=wobj_JMora;
        MoveL Target_8320,v60,z1,MarcadorVirtual\WObj:=wobj_JMora;
        MoveL Target_8330,v60,z1,MarcadorVirtual\WObj:=wobj_JMora;
        MoveL Target_8340,v60,z1,MarcadorVirtual\WObj:=wobj_JMora;
        MoveL Target_8350,v60,z1,MarcadorVirtual\WObj:=wobj_JMora;
        MoveL Target_8360,v60,z1,MarcadorVirtual\WObj:=wobj_JMora;
        MoveL Target_8370,v60,z1,MarcadorVirtual\WObj:=wobj_JMora;
        MoveL Target_8380,v60,z1,MarcadorVirtual\WObj:=wobj_JMora;
        MoveL Target_8390,v60,z1,MarcadorVirtual\WObj:=wobj_JMora;
        MoveL Target_8400,v60,z1,MarcadorVirtual\WObj:=wobj_JMora;
        MoveL Target_8410,v60,z1,MarcadorVirtual\WObj:=wobj_JMora;
        MoveL Target_8420,v60,z1,MarcadorVirtual\WObj:=wobj_JMora;
        MoveL Target_8430,v60,z1,MarcadorVirtual\WObj:=wobj_JMora;
        MoveL Target_8440,v60,z1,MarcadorVirtual\WObj:=wobj_JMora;
        MoveL Target_8450,v60,z1,MarcadorVirtual\WObj:=wobj_JMora;
        MoveL Target_8460,v60,z1,MarcadorVirtual\WObj:=wobj_JMora;
        MoveL Target_8470,v60,z1,MarcadorVirtual\WObj:=wobj_JMora;
        MoveL Target_8480,v60,z1,MarcadorVirtual\WObj:=wobj_JMora;
        MoveL Target_8490,v60,z1,MarcadorVirtual\WObj:=wobj_JMora;
        MoveL Target_8500,v60,z1,MarcadorVirtual\WObj:=wobj_JMora;
        MoveL Target_8510,v60,z1,MarcadorVirtual\WObj:=wobj_JMora;
        MoveL Target_8520,v60,z1,MarcadorVirtual\WObj:=wobj_JMora;
        MoveL Target_8530,v60,z1,MarcadorVirtual\WObj:=wobj_JMora;
        MoveL Target_8540,v60,z1,MarcadorVirtual\WObj:=wobj_JMora;
        MoveL Target_8550,v60,z1,MarcadorVirtual\WObj:=wobj_JMora;
        MoveL Target_8560,v60,z1,MarcadorVirtual\WObj:=wobj_JMora;
        MoveL Target_8570,v60,z1,MarcadorVirtual\WObj:=wobj_JMora;
        MoveL Target_8580,v60,z1,MarcadorVirtual\WObj:=wobj_JMora;
        MoveL Target_8590,v60,z1,MarcadorVirtual\WObj:=wobj_JMora;
        MoveL Target_8600,v60,z1,MarcadorVirtual\WObj:=wobj_JMora;
        MoveL Target_8610,v60,z1,MarcadorVirtual\WObj:=wobj_JMora;
        MoveL Target_8620,v60,z1,MarcadorVirtual\WObj:=wobj_JMora;
        MoveL Target_8630,v60,z1,MarcadorVirtual\WObj:=wobj_JMora;
        MoveL Target_8640,v60,z1,MarcadorVirtual\WObj:=wobj_JMora;
        MoveL Target_8650,v60,z1,MarcadorVirtual\WObj:=wobj_JMora;
        MoveL Target_8660,v60,z1,MarcadorVirtual\WObj:=wobj_JMora;
        MoveL Target_8670,v60,z1,MarcadorVirtual\WObj:=wobj_JMora;
        MoveL Target_8680,v60,z1,MarcadorVirtual\WObj:=wobj_JMora;
        MoveL Target_8690,v60,z1,MarcadorVirtual\WObj:=wobj_JMora;
        MoveL Target_8700,v60,z1,MarcadorVirtual\WObj:=wobj_JMora;
        MoveL Target_8710,v60,z1,MarcadorVirtual\WObj:=wobj_JMora;
        MoveL Target_8720,v60,z1,MarcadorVirtual\WObj:=wobj_JMora;
    ENDPROC
    PROC Path_cara()
        MoveL Target_8730,v60,z1,MarcadorVirtual\WObj:=wobj_JMora;
        MoveL Target_8740,v60,z1,MarcadorVirtual\WObj:=wobj_JMora;
        MoveL Target_8750,v60,z1,MarcadorVirtual\WObj:=wobj_JMora;
        MoveL Target_8760,v60,z1,MarcadorVirtual\WObj:=wobj_JMora;
        MoveL Target_8770,v60,z1,MarcadorVirtual\WObj:=wobj_JMora;
        MoveL Target_8780,v60,z1,MarcadorVirtual\WObj:=wobj_JMora;
        MoveL Target_8790,v60,z1,MarcadorVirtual\WObj:=wobj_JMora;
        MoveL Target_8800,v60,z1,MarcadorVirtual\WObj:=wobj_JMora;
        MoveL Target_8810,v60,z1,MarcadorVirtual\WObj:=wobj_JMora;
        MoveL Target_8820,v60,z1,MarcadorVirtual\WObj:=wobj_JMora;
        MoveL Target_8830,v60,z1,MarcadorVirtual\WObj:=wobj_JMora;
        MoveL Target_8840,v60,z1,MarcadorVirtual\WObj:=wobj_JMora;
        MoveL Target_8850,v60,z1,MarcadorVirtual\WObj:=wobj_JMora;
        MoveL Target_8860,v60,z1,MarcadorVirtual\WObj:=wobj_JMora;
        MoveL Target_8870,v60,z1,MarcadorVirtual\WObj:=wobj_JMora;
        MoveL Target_8880,v60,z1,MarcadorVirtual\WObj:=wobj_JMora;
        MoveL Target_8890,v60,z1,MarcadorVirtual\WObj:=wobj_JMora;
        MoveL Target_8900,v60,z1,MarcadorVirtual\WObj:=wobj_JMora;
        MoveL Target_8910,v60,z1,MarcadorVirtual\WObj:=wobj_JMora;
        MoveL Target_8920,v60,z1,MarcadorVirtual\WObj:=wobj_JMora;
        MoveL Target_8930,v60,z1,MarcadorVirtual\WObj:=wobj_JMora;
        MoveL Target_8940,v60,z1,MarcadorVirtual\WObj:=wobj_JMora;
        MoveL Target_8950,v60,z1,MarcadorVirtual\WObj:=wobj_JMora;
        MoveL Target_8960,v60,z1,MarcadorVirtual\WObj:=wobj_JMora;
        MoveL Target_8970,v60,z1,MarcadorVirtual\WObj:=wobj_JMora;
        MoveL Target_8980,v60,z1,MarcadorVirtual\WObj:=wobj_JMora;
        MoveL Target_8990,v60,z1,MarcadorVirtual\WObj:=wobj_JMora;
        MoveL Target_9000,v60,z1,MarcadorVirtual\WObj:=wobj_JMora;
        MoveL Target_9010,v60,z1,MarcadorVirtual\WObj:=wobj_JMora;
        MoveL Target_9020,v60,z1,MarcadorVirtual\WObj:=wobj_JMora;
        MoveL Target_9030,v60,z1,MarcadorVirtual\WObj:=wobj_JMora;
        MoveL Target_9040,v60,z1,MarcadorVirtual\WObj:=wobj_JMora;
        MoveL Target_9050,v60,z1,MarcadorVirtual\WObj:=wobj_JMora;
        MoveL Target_9060,v60,z1,MarcadorVirtual\WObj:=wobj_JMora;
        MoveL Target_9070,v60,z1,MarcadorVirtual\WObj:=wobj_JMora;
        MoveL Target_9080,v60,z1,MarcadorVirtual\WObj:=wobj_JMora;
        MoveL Target_9090,v60,z1,MarcadorVirtual\WObj:=wobj_JMora;
        MoveL Target_9100,v60,z1,MarcadorVirtual\WObj:=wobj_JMora;
        MoveL Target_9110,v60,z1,MarcadorVirtual\WObj:=wobj_JMora;
        MoveL Target_9120,v60,z1,MarcadorVirtual\WObj:=wobj_JMora;
        MoveL Target_9130,v60,z1,MarcadorVirtual\WObj:=wobj_JMora;
        MoveL Target_9140,v60,z1,MarcadorVirtual\WObj:=wobj_JMora;
        MoveL Target_9150,v60,z1,MarcadorVirtual\WObj:=wobj_JMora;
        MoveL Target_9160,v60,z1,MarcadorVirtual\WObj:=wobj_JMora;
        MoveL Target_9170,v60,z1,MarcadorVirtual\WObj:=wobj_JMora;
        MoveL Target_9180,v60,z1,MarcadorVirtual\WObj:=wobj_JMora;
        MoveL Target_9190,v60,z1,MarcadorVirtual\WObj:=wobj_JMora;
        MoveL Target_9200,v60,z1,MarcadorVirtual\WObj:=wobj_JMora;
        MoveL Target_9210,v60,z1,MarcadorVirtual\WObj:=wobj_JMora;
        MoveL Target_9220,v60,z1,MarcadorVirtual\WObj:=wobj_JMora;
        MoveL Target_9230,v60,z1,MarcadorVirtual\WObj:=wobj_JMora;
        MoveL Target_9240,v60,z1,MarcadorVirtual\WObj:=wobj_JMora;
        MoveL Target_9250,v60,z1,MarcadorVirtual\WObj:=wobj_JMora;
        MoveL Target_9260,v60,z1,MarcadorVirtual\WObj:=wobj_JMora;
        MoveL Target_9270,v60,z1,MarcadorVirtual\WObj:=wobj_JMora;
        MoveL Target_9280,v60,z1,MarcadorVirtual\WObj:=wobj_JMora;
        MoveL Target_9290,v60,z1,MarcadorVirtual\WObj:=wobj_JMora;
        MoveL Target_9300,v60,z1,MarcadorVirtual\WObj:=wobj_JMora;
        MoveL Target_9310,v60,z1,MarcadorVirtual\WObj:=wobj_JMora;
        MoveL Target_9320,v60,z1,MarcadorVirtual\WObj:=wobj_JMora;
        MoveL Target_9330,v60,z1,MarcadorVirtual\WObj:=wobj_JMora;
        MoveL Target_9340,v60,z1,MarcadorVirtual\WObj:=wobj_JMora;
        MoveL Target_9350,v60,z1,MarcadorVirtual\WObj:=wobj_JMora;
        MoveL Target_9360,v60,z1,MarcadorVirtual\WObj:=wobj_JMora;
        MoveL Target_9370,v60,z1,MarcadorVirtual\WObj:=wobj_JMora;
        MoveL Target_9380,v60,z1,MarcadorVirtual\WObj:=wobj_JMora;
        MoveL Target_9390,v60,z1,MarcadorVirtual\WObj:=wobj_JMora;
        MoveL Target_9400,v60,z1,MarcadorVirtual\WObj:=wobj_JMora;
        MoveL Target_9410,v60,z1,MarcadorVirtual\WObj:=wobj_JMora;
        MoveL Target_9420,v60,z1,MarcadorVirtual\WObj:=wobj_JMora;
        MoveL Target_9430,v60,z1,MarcadorVirtual\WObj:=wobj_JMora;
        MoveL Target_9440,v60,z1,MarcadorVirtual\WObj:=wobj_JMora;
        MoveL Target_9450,v60,z1,MarcadorVirtual\WObj:=wobj_JMora;
        MoveL Target_9460,v60,z1,MarcadorVirtual\WObj:=wobj_JMora;
        MoveL Target_9470,v60,z1,MarcadorVirtual\WObj:=wobj_JMora;
        MoveL Target_9480,v60,z1,MarcadorVirtual\WObj:=wobj_JMora;
        MoveL Target_9490,v60,z1,MarcadorVirtual\WObj:=wobj_JMora;
        MoveL Target_9500,v60,z1,MarcadorVirtual\WObj:=wobj_JMora;
        MoveL Target_9510,v60,z1,MarcadorVirtual\WObj:=wobj_JMora;
        MoveL Target_9520,v60,z1,MarcadorVirtual\WObj:=wobj_JMora;
        MoveL Target_9530,v60,z1,MarcadorVirtual\WObj:=wobj_JMora;
        MoveL Target_9540,v60,z1,MarcadorVirtual\WObj:=wobj_JMora;
        MoveL Target_9550,v60,z1,MarcadorVirtual\WObj:=wobj_JMora;
        MoveL Target_9560,v60,z1,MarcadorVirtual\WObj:=wobj_JMora;
        MoveL Target_9570,v60,z1,MarcadorVirtual\WObj:=wobj_JMora;
        MoveL Target_9580,v60,z1,MarcadorVirtual\WObj:=wobj_JMora;
        MoveL Target_9590,v60,z1,MarcadorVirtual\WObj:=wobj_JMora;
        MoveL Target_9600,v60,z1,MarcadorVirtual\WObj:=wobj_JMora;
        MoveL Target_9610,v60,z1,MarcadorVirtual\WObj:=wobj_JMora;
        MoveL Target_9620,v60,z1,MarcadorVirtual\WObj:=wobj_JMora;
        MoveL Target_9630,v60,z1,MarcadorVirtual\WObj:=wobj_JMora;
        MoveL Target_9640,v60,z1,MarcadorVirtual\WObj:=wobj_JMora;
        MoveL Target_9650,v60,z1,MarcadorVirtual\WObj:=wobj_JMora;
        MoveL Target_9660,v60,z1,MarcadorVirtual\WObj:=wobj_JMora;
        MoveL Target_9670,v60,z1,MarcadorVirtual\WObj:=wobj_JMora;
        MoveL Target_9680,v60,z1,MarcadorVirtual\WObj:=wobj_JMora;
        MoveL Target_9690,v60,z1,MarcadorVirtual\WObj:=wobj_JMora;
        MoveL Target_9700,v60,z1,MarcadorVirtual\WObj:=wobj_JMora;
        MoveL Target_9710,v60,z1,MarcadorVirtual\WObj:=wobj_JMora;
        MoveL Target_9720,v60,z1,MarcadorVirtual\WObj:=wobj_JMora;
        MoveL Target_9730,v60,z1,MarcadorVirtual\WObj:=wobj_JMora;
        MoveL Target_9740,v60,z1,MarcadorVirtual\WObj:=wobj_JMora;
        MoveL Target_9750,v60,z1,MarcadorVirtual\WObj:=wobj_JMora;
        MoveL Target_9760,v60,z1,MarcadorVirtual\WObj:=wobj_JMora;
        MoveL Target_9770,v60,z1,MarcadorVirtual\WObj:=wobj_JMora;
        MoveL Target_9780,v60,z1,MarcadorVirtual\WObj:=wobj_JMora;
        MoveL Target_9790,v60,z1,MarcadorVirtual\WObj:=wobj_JMora;
        MoveL Target_9800,v60,z1,MarcadorVirtual\WObj:=wobj_JMora;
        MoveL Target_9810,v60,z1,MarcadorVirtual\WObj:=wobj_JMora;
        MoveL Target_9820,v60,z1,MarcadorVirtual\WObj:=wobj_JMora;
        MoveL Target_9830,v60,z1,MarcadorVirtual\WObj:=wobj_JMora;
        MoveL Target_9840,v60,z1,MarcadorVirtual\WObj:=wobj_JMora;
        MoveL Target_9850,v60,z1,MarcadorVirtual\WObj:=wobj_JMora;
        MoveL Target_9860,v60,z1,MarcadorVirtual\WObj:=wobj_JMora;
        MoveL Target_9870,v60,z1,MarcadorVirtual\WObj:=wobj_JMora;
        MoveL Target_9880,v60,z1,MarcadorVirtual\WObj:=wobj_JMora;
        MoveL Target_9890,v60,z1,MarcadorVirtual\WObj:=wobj_JMora;
        MoveL Target_9900,v60,z1,MarcadorVirtual\WObj:=wobj_JMora;
        MoveL Target_9910,v60,z1,MarcadorVirtual\WObj:=wobj_JMora;
        MoveL Target_9920,v60,z1,MarcadorVirtual\WObj:=wobj_JMora;
        MoveL Target_9930,v60,z1,MarcadorVirtual\WObj:=wobj_JMora;
        MoveL Target_9940,v60,z1,MarcadorVirtual\WObj:=wobj_JMora;
        MoveL Target_9950,v60,z1,MarcadorVirtual\WObj:=wobj_JMora;
        MoveL Target_9960,v60,z1,MarcadorVirtual\WObj:=wobj_JMora;
        MoveL Target_9970,v60,z1,MarcadorVirtual\WObj:=wobj_JMora;
        MoveL Target_9980,v60,z1,MarcadorVirtual\WObj:=wobj_JMora;
        MoveL Target_9990,v60,z1,MarcadorVirtual\WObj:=wobj_JMora;
        MoveL Target_10000,v60,z1,MarcadorVirtual\WObj:=wobj_JMora;
        MoveL Target_10010,v60,z1,MarcadorVirtual\WObj:=wobj_JMora;
        MoveL Target_10020,v60,z1,MarcadorVirtual\WObj:=wobj_JMora;
        MoveL Target_10030,v60,z1,MarcadorVirtual\WObj:=wobj_JMora;
        MoveL Target_10040,v60,z1,MarcadorVirtual\WObj:=wobj_JMora;
        MoveL Target_10050,v60,z1,MarcadorVirtual\WObj:=wobj_JMora;
        MoveL Target_10060,v60,z1,MarcadorVirtual\WObj:=wobj_JMora;
        MoveL Target_10070,v60,z1,MarcadorVirtual\WObj:=wobj_JMora;
        MoveL Target_10080,v60,z1,MarcadorVirtual\WObj:=wobj_JMora;
        MoveL Target_10090,v60,z1,MarcadorVirtual\WObj:=wobj_JMora;
        MoveL Target_10100,v60,z1,MarcadorVirtual\WObj:=wobj_JMora;
        MoveL Target_10110,v60,z1,MarcadorVirtual\WObj:=wobj_JMora;
        MoveL Target_10120,v60,z1,MarcadorVirtual\WObj:=wobj_JMora;
        MoveL Target_10130,v60,z1,MarcadorVirtual\WObj:=wobj_JMora;
    ENDPROC
    PROC Path_ojo1()
        MoveL Target_10140,v60,z1,MarcadorVirtual\WObj:=wobj_JMora;
        MoveL Target_10150,v60,z1,MarcadorVirtual\WObj:=wobj_JMora;
        MoveL Target_10160,v60,z1,MarcadorVirtual\WObj:=wobj_JMora;
        MoveL Target_10170,v60,z1,MarcadorVirtual\WObj:=wobj_JMora;
        MoveL Target_10180,v60,z1,MarcadorVirtual\WObj:=wobj_JMora;
        MoveL Target_10190,v60,z1,MarcadorVirtual\WObj:=wobj_JMora;
        MoveL Target_10200,v60,z1,MarcadorVirtual\WObj:=wobj_JMora;
        MoveL Target_10210,v60,z1,MarcadorVirtual\WObj:=wobj_JMora;
        MoveL Target_10220,v60,z1,MarcadorVirtual\WObj:=wobj_JMora;
        MoveL Target_10230,v60,z1,MarcadorVirtual\WObj:=wobj_JMora;
        MoveL Target_10240,v60,z1,MarcadorVirtual\WObj:=wobj_JMora;
        MoveL Target_10250,v60,z1,MarcadorVirtual\WObj:=wobj_JMora;
        MoveL Target_10260,v60,z1,MarcadorVirtual\WObj:=wobj_JMora;
        MoveL Target_10270,v60,z1,MarcadorVirtual\WObj:=wobj_JMora;
        MoveL Target_10280,v60,z1,MarcadorVirtual\WObj:=wobj_JMora;
        MoveL Target_10290,v60,z1,MarcadorVirtual\WObj:=wobj_JMora;
        MoveL Target_10300,v60,z1,MarcadorVirtual\WObj:=wobj_JMora;
        MoveL Target_10310,v60,z1,MarcadorVirtual\WObj:=wobj_JMora;
        MoveL Target_10320,v60,z1,MarcadorVirtual\WObj:=wobj_JMora;
        MoveL Target_10330,v60,z1,MarcadorVirtual\WObj:=wobj_JMora;
        MoveL Target_10340,v60,z1,MarcadorVirtual\WObj:=wobj_JMora;
        MoveL Target_10350,v60,z1,MarcadorVirtual\WObj:=wobj_JMora;
        MoveL Target_10360,v60,z1,MarcadorVirtual\WObj:=wobj_JMora;
        MoveL Target_10370,v60,z1,MarcadorVirtual\WObj:=wobj_JMora;
        MoveL Target_10380,v60,z1,MarcadorVirtual\WObj:=wobj_JMora;
        MoveL Target_10390,v60,z1,MarcadorVirtual\WObj:=wobj_JMora;
        MoveL Target_10400,v60,z1,MarcadorVirtual\WObj:=wobj_JMora;
        MoveL Target_10410,v60,z1,MarcadorVirtual\WObj:=wobj_JMora;
        MoveL Target_10420,v60,z1,MarcadorVirtual\WObj:=wobj_JMora;
        MoveL Target_10430,v60,z1,MarcadorVirtual\WObj:=wobj_JMora;
        MoveL Target_10440,v60,z1,MarcadorVirtual\WObj:=wobj_JMora;
        MoveL Target_10450,v60,z1,MarcadorVirtual\WObj:=wobj_JMora;
        MoveL Target_10460,v60,z1,MarcadorVirtual\WObj:=wobj_JMora;
        MoveL Target_10470,v60,z1,MarcadorVirtual\WObj:=wobj_JMora;
        MoveL Target_10480,v60,z1,MarcadorVirtual\WObj:=wobj_JMora;
        MoveL Target_10490,v60,z1,MarcadorVirtual\WObj:=wobj_JMora;
        MoveL Target_10500,v60,z1,MarcadorVirtual\WObj:=wobj_JMora;
        MoveL Target_10510,v60,z1,MarcadorVirtual\WObj:=wobj_JMora;
        MoveL Target_10520,v60,z1,MarcadorVirtual\WObj:=wobj_JMora;
        MoveL Target_10530,v60,z1,MarcadorVirtual\WObj:=wobj_JMora;
        MoveL Target_10540,v60,z1,MarcadorVirtual\WObj:=wobj_JMora;
        MoveL Target_10550,v60,z1,MarcadorVirtual\WObj:=wobj_JMora;
        MoveL Target_10560,v60,z1,MarcadorVirtual\WObj:=wobj_JMora;
        MoveL Target_10570,v60,z1,MarcadorVirtual\WObj:=wobj_JMora;
        MoveL Target_10580,v60,z1,MarcadorVirtual\WObj:=wobj_JMora;
        MoveL Target_10590,v60,z1,MarcadorVirtual\WObj:=wobj_JMora;
        MoveL Target_10600,v60,z1,MarcadorVirtual\WObj:=wobj_JMora;
        MoveL Target_10610,v60,z1,MarcadorVirtual\WObj:=wobj_JMora;
        MoveL Target_10620,v60,z1,MarcadorVirtual\WObj:=wobj_JMora;
        MoveL Target_10630,v60,z1,MarcadorVirtual\WObj:=wobj_JMora;
        MoveL Target_10640,v60,z1,MarcadorVirtual\WObj:=wobj_JMora;
        MoveL Target_10650,v60,z1,MarcadorVirtual\WObj:=wobj_JMora;
        MoveL Target_10660,v60,z1,MarcadorVirtual\WObj:=wobj_JMora;
        MoveL Target_10670,v60,z1,MarcadorVirtual\WObj:=wobj_JMora;
        MoveL Target_10680,v60,z1,MarcadorVirtual\WObj:=wobj_JMora;
        MoveL Target_10690,v60,z1,MarcadorVirtual\WObj:=wobj_JMora;
        MoveL Target_10700,v60,z1,MarcadorVirtual\WObj:=wobj_JMora;
        MoveL Target_10710,v60,z1,MarcadorVirtual\WObj:=wobj_JMora;
        MoveL Target_10720,v60,z1,MarcadorVirtual\WObj:=wobj_JMora;
        MoveL Target_10730,v60,z1,MarcadorVirtual\WObj:=wobj_JMora;
        MoveL Target_10740,v60,z1,MarcadorVirtual\WObj:=wobj_JMora;
        MoveL Target_10750,v60,z1,MarcadorVirtual\WObj:=wobj_JMora;
        MoveL Target_10760,v60,z1,MarcadorVirtual\WObj:=wobj_JMora;
        MoveL Target_10770,v60,z1,MarcadorVirtual\WObj:=wobj_JMora;
        MoveL Target_10780,v60,z1,MarcadorVirtual\WObj:=wobj_JMora;
        MoveL Target_10790,v60,z1,MarcadorVirtual\WObj:=wobj_JMora;
        MoveL Target_10800,v60,z1,MarcadorVirtual\WObj:=wobj_JMora;
        MoveL Target_10810,v60,z1,MarcadorVirtual\WObj:=wobj_JMora;
        MoveL Target_10820,v60,z1,MarcadorVirtual\WObj:=wobj_JMora;
        MoveL Target_10830,v60,z1,MarcadorVirtual\WObj:=wobj_JMora;
    ENDPROC
    PROC Path_ojo2()
        MoveL Target_10840,v60,z1,MarcadorVirtual\WObj:=wobj_JMora;
        MoveL Target_10850,v60,z1,MarcadorVirtual\WObj:=wobj_JMora;
        MoveL Target_10860,v60,z1,MarcadorVirtual\WObj:=wobj_JMora;
        MoveL Target_10870,v60,z1,MarcadorVirtual\WObj:=wobj_JMora;
        MoveL Target_10880,v60,z1,MarcadorVirtual\WObj:=wobj_JMora;
        MoveL Target_10890,v60,z1,MarcadorVirtual\WObj:=wobj_JMora;
        MoveL Target_10900,v60,z1,MarcadorVirtual\WObj:=wobj_JMora;
        MoveL Target_10910,v60,z1,MarcadorVirtual\WObj:=wobj_JMora;
        MoveL Target_10920,v60,z1,MarcadorVirtual\WObj:=wobj_JMora;
        MoveL Target_10930,v60,z1,MarcadorVirtual\WObj:=wobj_JMora;
        MoveL Target_10940,v60,z1,MarcadorVirtual\WObj:=wobj_JMora;
        MoveL Target_10950,v60,z1,MarcadorVirtual\WObj:=wobj_JMora;
        MoveL Target_10960,v60,z1,MarcadorVirtual\WObj:=wobj_JMora;
        MoveL Target_10970,v60,z1,MarcadorVirtual\WObj:=wobj_JMora;
        MoveL Target_10980,v60,z1,MarcadorVirtual\WObj:=wobj_JMora;
        MoveL Target_10990,v60,z1,MarcadorVirtual\WObj:=wobj_JMora;
        MoveL Target_11000,v60,z1,MarcadorVirtual\WObj:=wobj_JMora;
        MoveL Target_11010,v60,z1,MarcadorVirtual\WObj:=wobj_JMora;
        MoveL Target_11020,v60,z1,MarcadorVirtual\WObj:=wobj_JMora;
        MoveL Target_11030,v60,z1,MarcadorVirtual\WObj:=wobj_JMora;
        MoveL Target_11040,v60,z1,MarcadorVirtual\WObj:=wobj_JMora;
        MoveL Target_11050,v60,z1,MarcadorVirtual\WObj:=wobj_JMora;
        MoveL Target_11060,v60,z1,MarcadorVirtual\WObj:=wobj_JMora;
        MoveL Target_11070,v60,z1,MarcadorVirtual\WObj:=wobj_JMora;
        MoveL Target_11080,v60,z1,MarcadorVirtual\WObj:=wobj_JMora;
        MoveL Target_11090,v60,z1,MarcadorVirtual\WObj:=wobj_JMora;
        MoveL Target_11100,v60,z1,MarcadorVirtual\WObj:=wobj_JMora;
        MoveL Target_11110,v60,z1,MarcadorVirtual\WObj:=wobj_JMora;
        MoveL Target_11120,v60,z1,MarcadorVirtual\WObj:=wobj_JMora;
        MoveL Target_11130,v60,z1,MarcadorVirtual\WObj:=wobj_JMora;
        MoveL Target_11140,v60,z1,MarcadorVirtual\WObj:=wobj_JMora;
        MoveL Target_11150,v60,z1,MarcadorVirtual\WObj:=wobj_JMora;
        MoveL Target_11160,v60,z1,MarcadorVirtual\WObj:=wobj_JMora;
        MoveL Target_11170,v60,z1,MarcadorVirtual\WObj:=wobj_JMora;
        MoveL Target_11180,v60,z1,MarcadorVirtual\WObj:=wobj_JMora;
        MoveL Target_11190,v60,z1,MarcadorVirtual\WObj:=wobj_JMora;
        MoveL Target_11200,v60,z1,MarcadorVirtual\WObj:=wobj_JMora;
        MoveL Target_11210,v60,z1,MarcadorVirtual\WObj:=wobj_JMora;
        MoveL Target_11220,v60,z1,MarcadorVirtual\WObj:=wobj_JMora;
        MoveL Target_11230,v60,z1,MarcadorVirtual\WObj:=wobj_JMora;
        MoveL Target_11240,v60,z1,MarcadorVirtual\WObj:=wobj_JMora;
        MoveL Target_11250,v60,z1,MarcadorVirtual\WObj:=wobj_JMora;
        MoveL Target_11260,v60,z1,MarcadorVirtual\WObj:=wobj_JMora;
        MoveL Target_11270,v60,z1,MarcadorVirtual\WObj:=wobj_JMora;
        MoveL Target_11280,v60,z1,MarcadorVirtual\WObj:=wobj_JMora;
        MoveL Target_11290,v60,z1,MarcadorVirtual\WObj:=wobj_JMora;
        MoveL Target_11300,v60,z1,MarcadorVirtual\WObj:=wobj_JMora;
        MoveL Target_11310,v60,z1,MarcadorVirtual\WObj:=wobj_JMora;
        MoveL Target_11320,v60,z1,MarcadorVirtual\WObj:=wobj_JMora;
        MoveL Target_11330,v60,z1,MarcadorVirtual\WObj:=wobj_JMora;
        MoveL Target_11340,v60,z1,MarcadorVirtual\WObj:=wobj_JMora;
        MoveL Target_11350,v60,z1,MarcadorVirtual\WObj:=wobj_JMora;
        MoveL Target_11360,v60,z1,MarcadorVirtual\WObj:=wobj_JMora;
        MoveL Target_11370,v60,z1,MarcadorVirtual\WObj:=wobj_JMora;
        MoveL Target_11380,v60,z1,MarcadorVirtual\WObj:=wobj_JMora;
        MoveL Target_11390,v60,z1,MarcadorVirtual\WObj:=wobj_JMora;
        MoveL Target_11400,v60,z1,MarcadorVirtual\WObj:=wobj_JMora;
        MoveL Target_11410,v60,z1,MarcadorVirtual\WObj:=wobj_JMora;
        MoveL Target_11420,v60,z1,MarcadorVirtual\WObj:=wobj_JMora;
        MoveL Target_11430,v60,z1,MarcadorVirtual\WObj:=wobj_JMora;
        MoveL Target_11440,v60,z1,MarcadorVirtual\WObj:=wobj_JMora;
        MoveL Target_11450,v60,z1,MarcadorVirtual\WObj:=wobj_JMora;
        MoveL Target_11460,v60,z1,MarcadorVirtual\WObj:=wobj_JMora;
        MoveL Target_11470,v60,z1,MarcadorVirtual\WObj:=wobj_JMora;
        MoveL Target_11480,v60,z1,MarcadorVirtual\WObj:=wobj_JMora;
        MoveL Target_11490,v60,z1,MarcadorVirtual\WObj:=wobj_JMora;
        MoveL Target_11500,v60,z1,MarcadorVirtual\WObj:=wobj_JMora;
        MoveL Target_11510,v60,z1,MarcadorVirtual\WObj:=wobj_JMora;
        MoveL Target_11520,v60,z1,MarcadorVirtual\WObj:=wobj_JMora;
        MoveL Target_11530,v60,z1,MarcadorVirtual\WObj:=wobj_JMora;
    ENDPROC
    PROC Path_boca1()
        MoveL Target_11540,v60,z1,MarcadorVirtual\WObj:=wobj_JMora;
        MoveL Target_11550,v60,z1,MarcadorVirtual\WObj:=wobj_JMora;
        MoveL Target_11560,v60,z1,MarcadorVirtual\WObj:=wobj_JMora;
        MoveL Target_11570,v60,z1,MarcadorVirtual\WObj:=wobj_JMora;
        MoveL Target_11580,v60,z1,MarcadorVirtual\WObj:=wobj_JMora;
        MoveL Target_11590,v60,z1,MarcadorVirtual\WObj:=wobj_JMora;
        MoveL Target_11600,v60,z1,MarcadorVirtual\WObj:=wobj_JMora;
    ENDPROC
    PROC Path_boca2()
        MoveL Target_11610,v60,z1,MarcadorVirtual\WObj:=wobj_JMora;
        MoveL Target_11620,v60,z1,MarcadorVirtual\WObj:=wobj_JMora;
        MoveL Target_11630,v60,z1,MarcadorVirtual\WObj:=wobj_JMora;
        MoveL Target_11640,v60,z1,MarcadorVirtual\WObj:=wobj_JMora;
        MoveL Target_11650,v60,z1,MarcadorVirtual\WObj:=wobj_JMora;
        MoveL Target_11660,v60,z1,MarcadorVirtual\WObj:=wobj_JMora;
        MoveL Target_11670,v60,z1,MarcadorVirtual\WObj:=wobj_JMora;
    ENDPROC
    PROC Path_boca3()
        MoveL Target_11680,v60,z1,MarcadorVirtual\WObj:=wobj_JMora;
        MoveL Target_11690,v60,z1,MarcadorVirtual\WObj:=wobj_JMora;
        MoveL Target_11700,v60,z1,MarcadorVirtual\WObj:=wobj_JMora;
        MoveL Target_11710,v60,z1,MarcadorVirtual\WObj:=wobj_JMora;
        MoveL Target_11720,v60,z1,MarcadorVirtual\WObj:=wobj_JMora;
        MoveL Target_11730,v60,z1,MarcadorVirtual\WObj:=wobj_JMora;
        MoveL Target_11740,v60,z1,MarcadorVirtual\WObj:=wobj_JMora;
    ENDPROC
    PROC Path_70()
        MoveL Target_2660,v60,z1,MarcadorVirtual\WObj:=wobj_JMora;
        MoveL Target_2670,v60,z1,MarcadorVirtual\WObj:=wobj_JMora;
    ENDPROC
    PROC Path_80()
        MoveL Target_3130,v60,z1,MarcadorVirtual\WObj:=wobj_JMora;
        MoveL Target_3140,v60,z1,MarcadorVirtual\WObj:=wobj_JMora;
    ENDPROC
    PROC Path_90()
        MoveL Target_3820,v60,z1,MarcadorVirtual\WObj:=wobj_JMora;
        MoveL Target_3830,v60,z1,MarcadorVirtual\WObj:=wobj_JMora;
    ENDPROC
    PROC Path_100()
        MoveL Target_4250,v60,z1,MarcadorVirtual\WObj:=wobj_JMora;
        MoveL Target_4260,v60,z1,MarcadorVirtual\WObj:=wobj_JMora;
    ENDPROC
    PROC Path_110()
        MoveL Target_5050,v60,z1,MarcadorVirtual\WObj:=wobj_JMora;
        MoveL Target_5060,v60,z1,MarcadorVirtual\WObj:=wobj_JMora;
    ENDPROC
    PROC Path_120()
        MoveL Target_5930,v60,z1,MarcadorVirtual\WObj:=wobj_JMora;
        MoveL Target_5940,v60,z1,MarcadorVirtual\WObj:=wobj_JMora;
    ENDPROC
    PROC Path_130()
        MoveL Target_6390,v60,z1,MarcadorVirtual\WObj:=wobj_JMora;
        MoveL Target_6400,v60,z1,MarcadorVirtual\WObj:=wobj_JMora;
    ENDPROC
    PROC Path_140()
        MoveL Target_7330,v60,z1,MarcadorVirtual\WObj:=wobj_JMora;
        MoveL Target_7340,v60,z1,MarcadorVirtual\WObj:=wobj_JMora;
    ENDPROC
    PROC Path_150()
        MoveL Target_8000,v60,z1,MarcadorVirtual\WObj:=wobj_JMora;
        MoveL Target_8010,v60,z1,MarcadorVirtual\WObj:=wobj_JMora;
    ENDPROC

    PROC Path_160()
        MoveL Target_8720,v60,z1,MarcadorVirtual\WObj:=wobj_JMora;
        MoveL Target_8730,v60,z1,MarcadorVirtual\WObj:=wobj_JMora;
    ENDPROC

    PROC Path_170()
        MoveL Target_10130,v60,z1,MarcadorVirtual\WObj:=wobj_JMora;
        MoveL Target_10140,v60,z1,MarcadorVirtual\WObj:=wobj_JMora;
    ENDPROC
    PROC Path_180()
        MoveL Target_10830,v60,z1,MarcadorVirtual\WObj:=wobj_JMora;
        MoveL Target_10840,v60,z1,MarcadorVirtual\WObj:=wobj_JMora;
    ENDPROC
    PROC Path_190()
        MoveL Target_11530,v60,z1,MarcadorVirtual\WObj:=wobj_JMora;
        MoveL Target_11540,v60,z1,MarcadorVirtual\WObj:=wobj_JMora;
    ENDPROC
    PROC Path_200()
        MoveL Target_11600,v60,z1,MarcadorVirtual\WObj:=wobj_JMora;
        MoveL Target_11610,v60,z1,MarcadorVirtual\WObj:=wobj_JMora;
    ENDPROC
    PROC Path_210()
        MoveL Target_11670,v60,z1,MarcadorVirtual\WObj:=wobj_JMora;
        MoveL Target_11680,v60,z1,MarcadorVirtual\WObj:=wobj_JMora;
    ENDPROC
    PROC Path_220()
        MoveL Target_11740,v60,z1,MarcadorVirtual\WObj:=wobj_JMora;
        MoveL Target_aprox1,v60,z1,MarcadorVirtual\WObj:=wobj0;
    ENDPROC

    ! Si tienes otras rutinas creadas (ej. PROC Dibujar_Circulo),
    ! deben ir aquí abajo, antes del ENDMODULE.

ENDMODULE
